(* CODESYS project yaskawafunctions.library
   Company: Evolution
   Title: YaskawaFunctions
   Version: 1.0.0.0

Project tree, tasks and I/O mapping:
  libraries: Tc2_System, * (Beckhoff Automation GmbH); Tc2_Utilities, * (Beckhoff Automation GmbH); Tc2_EtherCAT, * (Beckhoff Automation GmbH); Tc2_Standard, * (Beckhoff Automation GmbH)
  Data types/
    data type E_AccessType
    data type E_AmpType
    data type E_AmpVers
    data type E_EepromType
    data type E_SpecialParameter
    data type E_ValueType
    data type E_WhenEnabled
    data type E_Y_FB_Version
    data type ST_SigmaObject
  Global Variables/
    global variables Constants
  POUs/
    function block Y_AbsoluteEncoderReset [ST]
    function block Y_StoreParameters [ST]
    function block Y_WriteParameters [ST]
  Visualizations/
*)

// Data types/E_AccessType
TYPE E_AccessType : (
	ACCESS_RO		:=0,
	ACCESS_RW	:=1
	);
END_TYPE

// Data types/E_AmpType
TYPE E_AmpType : (
	BOTH_ROT_LIN		:=0,
	ROTARY			:=1,
	LINEAR				:=2
	);
END_TYPE

// Data types/E_AmpVers
TYPE E_AmpVers : (
	VERS_1_0	:=1,
	VERS_2_0	:=2	(*Vers Up*)
	);
END_TYPE

// Data types/E_EepromType
TYPE E_EepromType : (
	EEPROM_NO	:=0,
	EEPROM_YES	:=1
	);
END_TYPE

// Data types/E_SpecialParameter
TYPE E_SpecialParameter : (
	NOTHING_SPECIAL										:=0,	(*	16#0000	*)
	CHANGE_ECAT_PREOP							 		:=1,	(*	16#0001	*)	(*This object can be changed only in the EtherCAT Pre-Operational state*)
	CONDITIONAL_OBJECT									:=2,	(*	16#0002	*)	(*This object has to be set after another object is set. Ex:1C12:01*)
	CHANGE_ECAT_PREOP_AND_IS_DEPENDENT				:=3,
	OBJECT_COMMAND										:=4,	(*	16#0004	*)	(*This object must be executed to enable new settings.  Ex:2700h*)
(*	OBJECT_COMMAND_AND_CHANGE_ECAT_PREOP			:=5,
	OBJECT_COMMAND_AND_IS_DEPENDENT					:=6,
	OBJECT_COMMAND_AND_CHANGE_ECAT_PREOP_AND_IS_DEPENDENT	:=7,
*)	CHANGE_ECAT_DISABLED								:=8,	(*	16#0008	*)	(*This object can be changed only in Switch on Dsiabled state.*)
(*	CHANGE_ECAT_DISABLED_AND_CHANGE_ECAT_PREOP	:=9
	...
*)	CHANGE_ECAT_DISABLED_AND_OBJECT_COMMAND		:=12,	(*	16#0008 OR 16#0004 = 16#000C*)
(*	...
*)	HAS_DEPENDENT										:=16,	(*	16#0010	*)
(*	...
*)	CHANGE_ECAT_PREOP_AND_HAS_DEPENDENT			:=17	(*	16#0010 OR 16#0001 = 16#0011*)	
(*	...
	FUTURE_ADDITION_A									:=32,	(*	16#0020	*)
	...
	FUTURE_ADDITION_B									:=64,	(*	16#0020	*)
	...
*)

	);
END_TYPE

// Data types/E_ValueType
TYPE E_ValueType : (
	TYPE_NOT_SPECIFIED	:=0,
	TYPE_SINT				:=1,
	TYPE_INT				:=2,
	TYPE_DINT				:=3,
	TYPE_USINT			:=4,
	TYPE_UINT				:=5,
	TYPE_UDINT			:=6,
	TYPE_STRING			:=7
	);
END_TYPE

// Data types/E_WhenEnabled
TYPE E_WhenEnabled : (
	ENABLED_IMMEDIATELY		:=0,
	ENABLED_AFTER_RESTART 	:=1,
	ENABLED_SPECIAL			:=2
	);
END_TYPE

// Data types/E_Y_FB_Version
TYPE E_Y_FB_Version : (
	Y_FB_VER_1_0	:=1,
	Y_FB_VER_2_0	:=2	(*Vers Up*)
	);
END_TYPE

// Data types/ST_SigmaObject
TYPE ST_SigmaObject :
STRUCT
	Index			: WORD;		(* Index *)
	SubIndex		: USINT;		(* sub index *)
	(*Data type = UDINT*)
	Access				: USINT;	 	(*ENUM: ACCESS_RW, ACCESS_RO*)
	Eeprom				: USINT;	 	(*ENUM: EEPROM_NO, EEPROM_YES*)
	ValueSint			: SINT;		(* Parameter Data *)
	ValueInt				: INT;		(* Parameter Data *)
	ValueDint			: DINT;		(* Parameter Data *)
	ValueUsint			: USINT;		(* Parameter Data *)
	ValueUint			: UINT;		(* Parameter Data *)
	ValueUdint			: UDINT;		(* Parameter Data *)
	ValueString			: STRING;	(* Parameter Data *)
	ValueType			: USINT;		(*Parameter Data Type*)
	WhenEnabled		: USINT;		(*ENUM: ENABLED_AFTER_RESTART, ENABLED_IMMEDIATELY*)
	AmpType			: USINT; 		(*ENUM: ROTARY, LINEAR, BOTH_ROT_LIN*)
	EnRestartPattern		: WORD;		(* Specifies which bits of the parameter data require restart when changed *)
	AmpVers			: USINT 		:= VERS_1_0;
	SpecialParameter		: DWORD;	(*allows up to 32 switches*)
	DependentValueUsint	: USINT;		(*0 in all cases for version 1, Ex: 1600, 1601...*)

END_STRUCT
END_TYPE

// Global Variables/Constants
{attribute 'Tc2GvlVarNames'}
VAR_GLOBAL CONSTANT
	SAVE				:	UDINT		:=	16#65766173;		(*This is SAVE in ASCII with MSB leftmost, so that's EVAS*)
	USERPRMCFG		:	UDINT		:=	1;
	REVISION_1			:	UDINT		:=	16#00010000;
	REVISION_2			:	UDINT		:=	16#00020000;		(*Vers Up*)
	VENDOR_YASKAWA	:	UDINT		:=	16#00000539;
	PRODUCT_ROTARY	:	UDINT		:=	16#02200001;
	PRODUCT_LINEAR	:	UDINT		:=	16#02200002;
	SEND_REQUEST_1008	:	ARRAY [1..16] OF USINT	:=[	0,0,1,2,00,16#20,0,0,16#08,16#10,0,0,0,0,0,0];
	SEND_REQUEST_100E	:	ARRAY [1..16] OF USINT	:=[	0,0,1,2,00,16#20,0,0,16#0E,16#10,0,0,0,0,0,0];
	SEND_REQUEST_1013	:	ARRAY [1..16] OF USINT	:=[	0,0,1,2,00,16#20,0,0,16#13,16#10,0,0,0,0,0,0];
	SEND_PREPARATION	:	ARRAY [1..16] OF USINT		:=[	0,0,1,2,01,16#20,0,0,16#02,16#00,0,0,0,0,0,0];
	SEND_EXECUTE			:	ARRAY [1..16] OF USINT	:=[	0,0,1,2,01,16#20,0,0,16#01,16#00,0,0,0,0,0,0];
	SEND_ABORT			:	ARRAY [1..16] OF USINT	:=[	0,0,1,2,00,16#20,0,0,16#00,16#00,0,0,0,0,0,0];
END_VAR
VAR_GLOBAL
END_VAR

// POUs/Y_AbsoluteEncoderReset
FUNCTION_BLOCK Y_AbsoluteEncoderReset
VAR_INPUT
	bExecute		:	BOOL		;
	sNetId			:	T_AmsNetId	;
	nSlaveAddr 		:	UINT		;
END_VAR
VAR_OUTPUT
	bDone		:	BOOL			;
	bBusy		:	BOOL			;
	bError		:	BOOL			;
	nErrorID		:	UDINT			;
END_VAR
VAR
(*Extra Features Var Out*)
	sErrorString	:	T_MaxString		;
(*Internal variables*)
	State				:	UINT		:= 	0;
	VendorID			: 	UDINT		;
	ProductCode			: 	UDINT		;
	bNotExecute			:	BOOL		;
	StatusWord			: 	UINT		;
	nErrorIDRead			:	UDINT		;
	sNetIdRead			:	T_AmsNetId	;
	nSlaveAddrRead		:	UINT		;
	StatusAdjusting		:	USINT		;

(*Internal Function Blocks*)
	fbRisingEdge			: 	R_TRIG	;
	fbFallingEdge		: 	F_TRIG	;
	fbSdoReadEx		: 	FB_EcCoESdoReadEx 	:= (bExecute := FALSE, bCompleteAccess := FALSE);
	fbSdoWriteEx			:	FB_EcCoESdoWriteEx 	:= (bExecute := FALSE, bCompleteAccess := FALSE);
END_VAR

fbFallingEdge	(CLK:= bExecute);
IF fbFallingEdge.Q THEN
	bNotExecute	:=	TRUE;
END_IF;

(* Done is TRUE for one cycle when falling edge of Execute has occured *)
IF bDone AND bNotExecute THEN
	bDone		:=	FALSE;
END_IF;

IF bError AND bNotExecute THEN
	bError				:=	FALSE;
	nErrorId				:=	0;
	nErrorIDRead			:=	0;
END_IF;

CASE State OF
0:
fbRisingEdge		(CLK:= bExecute);
IF fbRisingEdge.Q THEN
	bDone				:=	FALSE;
	bBusy				:=	TRUE;
	bError				:=	FALSE;
	nErrorId				:=	0;
	nErrorIDRead			:=	0;
	sErrorString			:=	'';
	bNotExecute			:=	FALSE;
	sNetIdRead			:=	sNetId;
	nSlaveAddrRead		:=	nSlaveAddr;
	State				:=	10;
END_IF

1:
fbSdoReadEx(
	sNetId		:=	sNetIdRead,
	nSlaveAddr	:=	nSlaveAddrRead,
	nIndex		:=	16#1018,
	nSubIndex	:=	1,				(*Vendor ID*)
	pDstBuf		:=	ADR(VendorID),
	cbBufLen	:=	SIZEOF(VendorID),
	bExecute	:=	TRUE	);
State:=2;

2: (*SDO read, Read ID*)
fbSdoReadEx();
IF NOT fbSdoReadEx.bBusy THEN
	IF NOT fbSdoReadEx.bError THEN
		fbSdoReadEx(bExecute:= FALSE);
		State:=3;
		IF NOT (VendorID=VENDOR_YASKAWA) THEN 			(*Vendor ID = Yaskawa*)
			sErrorString:=CONCAT(CONCAT(
				'Product not compatible.  This FB is only for Vendor ID 0x00000539 (Yaskawa).  Vendor ID read as ',
				UDINT_TO_STRING(VendorID)),
				'.  ErrorID from FB, not from ADS.'
			);
			nErrorIDRead:=4100;
			State:=99;
		END_IF
	ELSE
		sErrorString:=CONCAT(CONCAT(
			'Error reading Product Code, Object: ',
			WORD_TO_STRING(fbSdoReadEx.nIndex)),
			'.  Perhaps the Axis Address or NetID is incorrect.  Error occurred using Function Block FB_EcCoESdoReadEx.  ErrorID is from FB_EcCoESdoReadEx.'
		);
		nErrorIDRead:=fbSdoReadEx.nErrId;
		State:=99;
	END_IF
END_IF

3: (*Read the product code*)
fbSdoReadEx(
	nSubIndex	:=	2,				(*Product Code*)
	pDstBuf		:=	ADR(ProductCode),
	cbBufLen	:=	SIZEOF(ProductCode),
	bExecute	:=	TRUE);
State:=4;

4: (*SDO read, Read ID*)
fbSdoReadEx();
IF NOT fbSdoReadEx.bBusy THEN
	IF NOT fbSdoReadEx.bError THEN
		fbSdoReadEx(bExecute:= FALSE);
		IF ProductCode=PRODUCT_ROTARY OR ProductCode=PRODUCT_LINEAR THEN 			(*Rotary Motor Detected*)
			State:=10;
		ELSE 									 (*neither Linear nor Rotary Motor Detected*)
			sErrorString:=CONCAT(CONCAT(
				'Product not compatible.  This FB is only for Product codes 0x02200001 (Sigma-5 Rotary) and 0x02200002 (Sigma-5 Linear).  If using Sigma-5 CoE Drive, get latest FB from Yaskawa.com.  Product code read as ',
				UDINT_TO_STRING(ProductCode)),
				'.  ErrorID from FB, not from ADS.'
			);
			nErrorIDRead:=4101;
			State:=99;
		END_IF
	ELSE
		sErrorString:=CONCAT(CONCAT(
			'Error reading Product Code, Object: ',
			WORD_TO_STRING(fbSdoReadEx.nIndex)),
			'.  Error occurred using Function Block FB_EcCoESdoReadEx.  ErrorID is from FB_EcCoESdoReadEx.'
		);
		nErrorIDRead:=fbSdoReadEx.nErrId;
		State:=99;
	END_IF
END_IF

10: (*check conditions for Absolute Reset - check for servo off - doesn't matter the encoder type, since incremental cannot be checked through ECAT*)
fbSdoReadEx( 			(*Get StatusWord*)
	sNetId		:= sNetIdRead,
	nSlaveAddr	:= nSlaveAddrRead ,
	nSubIndex	:= 0,
	nIndex		:= 16#6041,
	pDstBuf		:= ADR(StatusWord),
	cbBufLen	:= SIZEOF(StatusWord),
	bExecute	:= TRUE 		); (*rising edge required*)
State:=11;

11: (*Read the statusword to verify correct state for sending the adjusting command*)
fbSdoReadEx();
IF NOT fbSdoReadEx.bBusy THEN
	IF NOT fbSdoReadEx.bError THEN
		fbSdoReadEx(bExecute:= FALSE);
		IF
			NOT((UINT_TO_WORD(StatusWord) AND 2#0000_0000_0110_1111)=2#0000_0000_0000_0111) (*NOT Quick stop active*)
			AND
			NOT((UINT_TO_WORD(StatusWord) AND 2#0000_0010_0111_1111)=2#0000_0010_0011_0111) (*NOT Operation enabled*)
			AND
			NOT((UINT_TO_WORD(StatusWord) AND 2#0000_0000_0100_1111)=2#0000_0000_0000_1111) (*NOT Fault reaction active*)
			THEN 	(*servo is off - Required specifically for absolute encoder reset*)
			fbSdoWriteEx( (*Initialize WriteEx*)
				sNetId		:= sNetIdRead,
				nSlaveAddr	:= nSlaveAddrRead,
				bExecute	:= FALSE	); (*Second time initialized - first time was in declarations; maybe this line can be removed*)
			State:=12;
		ELSE
			sErrorString:=CONCAT(CONCAT(
				'Servo is on. StatusWord cannot be x00x_0111(bin), xx1x_x011_0111(bin), or x0xx_1111(bin), but read as ',
				UDINT_TO_STRING(StatusWord)),
				'(dec).  ErrorID from FB, not from ADS.'
			);
			nErrorIDRead:=4110;
			State:=99;
		END_IF
	ELSE
		sErrorString:=CONCAT(CONCAT(
			'Error reading StatusWord, Object: ',
			WORD_TO_STRING(fbSdoReadEx.nIndex)),
			'.  Error occurred using Function Block FB_EcCoESdoReadEx.  ErrorID is from FB_EcCoESdoReadEx.'
		);
		nErrorIDRead:=fbSdoReadEx.nErrId;
		State:=99;
	END_IF
END_IF

12: (*Send the data for the Request*)
fbSdoWriteEx(
	nIndex		:= 16#2710,
	nSubIndex	:= 1,
	pSrcBuf		:= ADR(SEND_REQUEST_1008), (*Absolute encoder reset*)
	cbBufLen	:= SIZEOF(SEND_REQUEST_1008),
	bExecute	:= TRUE);
State:=13;

13: (*Complete sending the request*)
fbSdoWriteEx();
IF NOT fbSdoWriteEx.bBusy THEN
	IF NOT fbSdoWriteEx.bError THEN
		fbSdoWriteEx(bExecute:= FALSE);
		State:=14;
	ELSE
		sErrorString:='Error sending Absolute Encoder Reset request to object 2710.  Error occurred using Function Block FB_EcCoESdoWriteEx.  ErrorID is from FB_EcCoESdoWriteEx.';
		nErrorIDRead:=fbSdoWriteEx.nErrId;
		State:=99;
	END_IF
END_IF

14:
fbSdoReadEx( 			(*Get Status (from 2710:02 USINT)*)
	nSubIndex	:= 2,
	nIndex		:= 16#2710,
	pDstBuf		:= ADR(StatusAdjusting),
	cbBufLen	:= SIZEOF(StatusAdjusting),
	bExecute	:= TRUE);
State:=15;

15: (*Read the Status to determine which state to perform next*)
fbSdoReadEx();
IF NOT fbSdoReadEx.bBusy THEN
	IF NOT fbSdoReadEx.bError THEN
		fbSdoReadEx(bExecute:= FALSE);
		CASE StatusAdjusting OF
			1:
				State:=20;
			2:	(*Error. Issue error, then issue Send Abort*)
				sErrorString:='Adjusting command: Send Request 1008 - failed.';
				nErrorIDRead:=4115;
				State:=50;
			3: 	(*Error. Read reply, Issue error, then issue Send Abort*)
				sErrorString:='Adjusting command: Send Request 1008 - failed.  Reply data exists in 0x2710:03.';
				nErrorIDRead:=4116;
				State:=50;
			255:
				State:=14;
			ELSE
				sErrorString:=CONCAT(CONCAT(
					'Status state is not valid (must be 1,2,3,255).  Read as ',
					UDINT_TO_STRING(StatusAdjusting)),
					'(dec).  ErrorID from FB, not from ADS.'
				);
				nErrorIDRead:=4111;
				State:=99;
			END_CASE
	ELSE
		sErrorString:='Error reading Adjusting Status, Object 2710:02.  Error occurred using Function Block FB_EcCoESdoReadEx.  ErrorID is from FB_EcCoESdoReadEx.';
		nErrorIDRead:=fbSdoReadEx.nErrId;
		State:=99;
	END_IF
END_IF

20: (*Continue with Step 2: Send the Preparation*)
(*Preparation is required for Absolute Encoder Reset*)
(*Send the data for the Preparation*)
fbSdoWriteEx(
	nIndex		:= 16#2710,
	nSubIndex	:= 1,
	pSrcBuf		:= ADR(SEND_PREPARATION),
	cbBufLen	:= SIZEOF(SEND_PREPARATION),
	bExecute	:= TRUE);
State:=21;

21: (*Complete sending the request*)
fbSdoWriteEx();
IF NOT fbSdoWriteEx.bBusy THEN
	IF NOT fbSdoWriteEx.bError THEN
		fbSdoWriteEx(bExecute:= FALSE);
		State:=22;
	ELSE
		sErrorString:='Error sending Preparation request to object 2710.  Error occurred using Function Block FB_EcCoESdoWriteEx.  ErrorID is from FB_EcCoESdoWriteEx.';
		nErrorIDRead:=fbSdoWriteEx.nErrId;
		State:=99;
	END_IF
END_IF

22:
fbSdoReadEx( 			(*Get Status (from 2710:02 USINT)*)
	nSubIndex	:= 2,
	nIndex		:= 16#2710,
	pDstBuf		:= ADR(StatusAdjusting),
	cbBufLen	:= SIZEOF(StatusAdjusting),
	bExecute	:= TRUE);
State:=23;

23: (*Read the Status to determine which state to perform next*)
fbSdoReadEx();
IF NOT fbSdoReadEx.bBusy THEN
	IF NOT fbSdoReadEx.bError THEN
		fbSdoReadEx(bExecute:= FALSE);
		CASE StatusAdjusting OF
			1:
				State:=30;
			2:	(*Error. Issue error, then issue Send Abort*)
				sErrorString:='Adjusting command: Send Preparation - failed.';
				nErrorIDRead:=4117;
				State:=50;
			3: 	(*Error. Read reply, Issue error, then issue Send Abort*)
				sErrorString:='Adjusting command: Send Preparation - failed.  Reply data exists in 0x2710:03.';
				nErrorIDRead:=4118;
				State:=50;
			255:
				State:=22;
			ELSE
				sErrorString:=CONCAT(CONCAT(
					'Status state is not valid (must be 1,2,3,255).  Read as ',
					UDINT_TO_STRING(StatusAdjusting)),
					'(dec).  ErrorID from FB, not from ADS.'
				);
				nErrorIDRead:=4111;
				State:=99;
			END_CASE
	ELSE
		sErrorString:='Error reading Adjusting Status, Object 2710:02.  Error occurred using Function Block FB_EcCoESdoReadEx.  ErrorID is from FB_EcCoESdoReadEx.';
		nErrorIDRead:=fbSdoReadEx.nErrId;
		State:=99;
	END_IF
END_IF

30: (*Continue with Step 2: Send the Execute*)
(*Send the data for the Execute*)
fbSdoWriteEx(
	nIndex		:= 16#2710,
	nSubIndex	:= 1,
	pSrcBuf		:= ADR(SEND_EXECUTE),
	cbBufLen	:= SIZEOF(SEND_EXECUTE),
	bExecute	:= TRUE);
State:=31;

31: (*Complete sending the request*)
fbSdoWriteEx();
IF NOT fbSdoWriteEx.bBusy THEN
	IF NOT fbSdoWriteEx.bError THEN
		fbSdoWriteEx(bExecute:= FALSE);
		State:=32;
	ELSE
		sErrorString:='Error sending Execute request to object 2710.  Error occurred using Function Block FB_EcCoESdoWriteEx.  ErrorID is from FB_EcCoESdoWriteEx.';
		nErrorIDRead:=fbSdoWriteEx.nErrId;
		State:=99;
	END_IF
END_IF

32:
fbSdoReadEx( 			(*Get Status (from 2710:02 USINT)*)
	nSubIndex	:= 2,
	nIndex		:= 16#2710,
	pDstBuf		:= ADR(StatusAdjusting),
	cbBufLen	:= SIZEOF(StatusAdjusting),
	bExecute	:= TRUE);
State:=33;

33: (*Read the Status to determine which state to perform next*)
fbSdoReadEx();
IF NOT fbSdoReadEx.bBusy THEN
	IF NOT fbSdoReadEx.bError THEN
		fbSdoReadEx(bExecute:= FALSE);
		CASE StatusAdjusting OF
			1:
				State:=40;
			2:	(*Error. Issue error, then issue Send Abort*)
				sErrorString:='Adjusting command: Send Execute - failed.';
				nErrorIDRead:=4119;
				State:=50;
			3: 	(*Error. Read reply, Issue error, then issue Send Abort*)
				sErrorString:='Adjusting command: Send Execute - failed.  Reply data exists in 0x2710:03.';
				nErrorIDRead:=4120;
				State:=50;
			255:
				State:=32;
			ELSE
				sErrorString:=CONCAT(CONCAT(
					'Status state is not valid (must be 1,2,3,255).  Read as ',
					UDINT_TO_STRING(StatusAdjusting)),
					'(dec).  ErrorID from FB, not from ADS.'
				);
				nErrorIDRead:=4111;
				State:=99;
			END_CASE
	ELSE
		sErrorString:='Error reading Adjusting Status, Object 2710:02.  Error occurred using Function Block FB_EcCoESdoReadEx.  ErrorID is from FB_EcCoESdoReadEx.';
		nErrorIDRead:=fbSdoReadEx.nErrId;
		State:=99;
	END_IF
END_IF

40: (*Finished Execution*)
	bDone	:=	TRUE;
	bBusy	:=	FALSE;
	State:=0;

50: (*Step 4: Send Abort (only applies if an error occurs)*)
fbSdoWriteEx(
	nIndex		:= 16#2710,
	nSubIndex	:= 1,
	pSrcBuf		:= ADR(SEND_ABORT),
	cbBufLen	:= SIZEOF(SEND_ABORT),
	bExecute	:= TRUE);
State:=51;

51: (*Complete sending the request*)
fbSdoWriteEx();
IF NOT fbSdoWriteEx.bBusy THEN
	IF NOT fbSdoWriteEx.bError THEN
		fbSdoWriteEx(bExecute:= FALSE);
		State:=52;
	ELSE
		sErrorString:='Error sending Abort request to object 2710.  Error occurred using Function Block FB_EcCoESdoWriteEx.  ErrorID is from FB_EcCoESdoWriteEx.  Also, error occurred performing Adjusting command, but ErrorID of this second error cannot be provided.';
		nErrorIDRead:=fbSdoWriteEx.nErrId;
		State:=99;
	END_IF
END_IF

52:
fbSdoReadEx( 			(*Get Status (from 2710:02 USINT)*)
	nSubIndex	:= 2,
	nIndex		:= 16#2710,
	pDstBuf		:= ADR(StatusAdjusting),
	cbBufLen	:= SIZEOF(StatusAdjusting),
	bExecute	:= TRUE);
State:=53;

53: (*Read the Status to determine which state to perform next*)
fbSdoReadEx();
IF NOT fbSdoReadEx.bBusy THEN
	IF NOT fbSdoReadEx.bError THEN
		fbSdoReadEx(bExecute:= FALSE);
		CASE StatusAdjusting OF
			1:
				sErrorString:=CONCAT(
				sErrorString,  (*Concatenate with error string from previous error state.*)
				'  Abort succeeded, but requested adjusting command failed.  ErrorID is from FB, not from ADS.'
				);
				State:=99;
			2:
				sErrorString:='Abort failed, and requested adjusting command failed.  ErrorID is from FB, not from ADS.';
				nErrorIDRead:=4113;
				State:=99;
			3:
				sErrorString:='Abort failed, and requested adjusting command failed.  Reply data exists in 0x2710:03.  ErrorID is from FB, not from ADS.';
				nErrorIDRead:=4114;
				State:=99;
			255:
				State:=52;
			ELSE
				sErrorString:=CONCAT(CONCAT(
					'Status state is not valid (must be 1,2,3,255).  Read as ',
					UDINT_TO_STRING(StatusAdjusting)),
					'(dec).  ErrorID from FB, not from ADS.  Also, error occurred performing Adjusting command, but ErrorID of this second error cannot be provided.'
				);
				nErrorIDRead:=4111;
				State:=99;
			END_CASE
	ELSE
		sErrorString:='Error reading Adjusting Status, Object 2710:02.  Error occurred using Function Block FB_EcCoESdoReadEx.  ErrorID is from FB_EcCoESdoReadEx.  Also, error occurred performing Adjusting command, but ErrorID of this second error cannot be provided.';
		nErrorIDRead:=fbSdoReadEx.nErrId;
		State:=99;
	END_IF
END_IF

99: (*Error State*)
	bBusy	:=	FALSE;
	bError	:=	TRUE;
	nErrorID	:=	nErrorIDRead;
	State	:=	0;

ELSE
	sErrorString:=CONCAT(CONCAT(
		'Internal function block error.  Function block state not found.  State read as: ',
		UINT_TO_STRING(State)),
		'.  ErrorID from FB, not from ADS.'
	);
	nErrorIDRead:=4112;
	State:=99;
END_CASE

END_FUNCTION_BLOCK

// POUs/Y_StoreParameters
FUNCTION_BLOCK Y_StoreParameters
VAR_INPUT
	bExecute		:	BOOL		;
	sNetId			:	T_AmsNetId	;
	nSlaveAddr 		:	UINT		;
	sFile			:	T_MaxString	:=	'C:\YaskawaPrm.dat' ;
END_VAR
VAR_OUTPUT
	bDone		:	BOOL			;
	bBusy		:	BOOL			;
	bError		:	BOOL			;
	nErrorID		:	UDINT			;
END_VAR
VAR
	(*Extra Features Var In*)
	bBypassCheck	:	BOOL		:=	FALSE;					(*Used to skip Version check, but not Vendor ID nor Product Code*)
	bBypassAutoFile	:	BOOL		:=	TRUE;
	sFileAuto		:	T_MaxString	:=	'C:\YaskawaPrm_'	; (*Time stamp and .dat is appended to this file name*)
	(*Extra Features Var Out*)
	sErrorString	:	T_MaxString		;

	AllSigmaObjects : ARRAY [1..364] OF ST_SigmaObject:=[
(*1*)		(Index:=16#1000,	SubIndex:=0,		ValueType:=TYPE_UDINT,		Access:=ACCESS_RO,		Eeprom:=EEPROM_NO,	AmpType:=BOTH_ROT_LIN,	WhenEnabled:=ENABLED_IMMEDIATELY),
		(Index:=16#1001,	SubIndex:=0,		ValueType:=TYPE_USINT,		Access:=ACCESS_RO,		Eeprom:=EEPROM_NO,	AmpType:=BOTH_ROT_LIN,	WhenEnabled:=ENABLED_IMMEDIATELY),
		(Index:=16#1008,	SubIndex:=0,		ValueType:=TYPE_STRING,	Access:=ACCESS_RO,		Eeprom:=EEPROM_NO,	AmpType:=BOTH_ROT_LIN,	WhenEnabled:=ENABLED_IMMEDIATELY),
		(Index:=16#100A,	SubIndex:=0,		ValueType:=TYPE_STRING,	Access:=ACCESS_RO,		Eeprom:=EEPROM_NO,	AmpType:=BOTH_ROT_LIN,	WhenEnabled:=ENABLED_IMMEDIATELY),
		(Index:=16#1010,	SubIndex:=0,		ValueType:=TYPE_USINT,		Access:=ACCESS_RO,		Eeprom:=EEPROM_NO,	AmpType:=BOTH_ROT_LIN,	WhenEnabled:=ENABLED_IMMEDIATELY),
		(Index:=16#1010,	SubIndex:=1,		ValueType:=TYPE_UDINT,		Access:=ACCESS_RW,	Eeprom:=EEPROM_NO,	AmpType:=BOTH_ROT_LIN,	WhenEnabled:=ENABLED_IMMEDIATELY,		SpecialParameter:=CHANGE_ECAT_DISABLED_AND_OBJECT_COMMAND),
		(Index:=16#1010,	SubIndex:=2,		ValueType:=TYPE_UDINT,		Access:=ACCESS_RW,	Eeprom:=EEPROM_NO,	AmpType:=BOTH_ROT_LIN,	WhenEnabled:=ENABLED_IMMEDIATELY,		SpecialParameter:=OBJECT_COMMAND),
		(Index:=16#1010,	SubIndex:=3,		ValueType:=TYPE_UDINT,		Access:=ACCESS_RW,	Eeprom:=EEPROM_NO,	AmpType:=BOTH_ROT_LIN,	WhenEnabled:=ENABLED_IMMEDIATELY,		SpecialParameter:=OBJECT_COMMAND),
		(Index:=16#1010,	SubIndex:=4,		ValueType:=TYPE_UDINT,		Access:=ACCESS_RW,	Eeprom:=EEPROM_NO,	AmpType:=BOTH_ROT_LIN,	WhenEnabled:=ENABLED_IMMEDIATELY,		SpecialParameter:=CHANGE_ECAT_DISABLED_AND_OBJECT_COMMAND),
(*10*)	(Index:=16#1011,	SubIndex:=0,		ValueType:=TYPE_USINT,		Access:=ACCESS_RO,		Eeprom:=EEPROM_NO,	AmpType:=BOTH_ROT_LIN,	WhenEnabled:=ENABLED_IMMEDIATELY),
		(Index:=16#1011,	SubIndex:=1,		ValueType:=TYPE_UDINT,		Access:=ACCESS_RW,	Eeprom:=EEPROM_NO,	AmpType:=BOTH_ROT_LIN,	WhenEnabled:=ENABLED_IMMEDIATELY,		SpecialParameter:=CHANGE_ECAT_DISABLED_AND_OBJECT_COMMAND),
		(Index:=16#1011,	SubIndex:=2,		ValueType:=TYPE_UDINT,		Access:=ACCESS_RW,	Eeprom:=EEPROM_NO,	AmpType:=BOTH_ROT_LIN,	WhenEnabled:=ENABLED_IMMEDIATELY,		SpecialParameter:=OBJECT_COMMAND),
		(Index:=16#1011,	SubIndex:=3,		ValueType:=TYPE_UDINT,		Access:=ACCESS_RW,	Eeprom:=EEPROM_NO,	AmpType:=BOTH_ROT_LIN,	WhenEnabled:=ENABLED_IMMEDIATELY,		SpecialParameter:=OBJECT_COMMAND),
		(Index:=16#1011,	SubIndex:=4,		ValueType:=TYPE_UDINT,		Access:=ACCESS_RW,	Eeprom:=EEPROM_NO,	AmpType:=BOTH_ROT_LIN,	WhenEnabled:=ENABLED_IMMEDIATELY,		SpecialParameter:=CHANGE_ECAT_DISABLED_AND_OBJECT_COMMAND),
		(Index:=16#1018,	SubIndex:=0,		ValueType:=TYPE_USINT,		Access:=ACCESS_RO,		Eeprom:=EEPROM_NO,	AmpType:=BOTH_ROT_LIN,	WhenEnabled:=ENABLED_IMMEDIATELY),
		(Index:=16#1018,	SubIndex:=1,		ValueType:=TYPE_UDINT,		Access:=ACCESS_RO,		Eeprom:=EEPROM_NO,	AmpType:=BOTH_ROT_LIN,	WhenEnabled:=ENABLED_IMMEDIATELY),
		(Index:=16#1018,	SubIndex:=2,		ValueType:=TYPE_UDINT,		Access:=ACCESS_RO,		Eeprom:=EEPROM_NO,	AmpType:=BOTH_ROT_LIN,	WhenEnabled:=ENABLED_IMMEDIATELY),
		(Index:=16#1018,	SubIndex:=3,		ValueType:=TYPE_UDINT,		Access:=ACCESS_RO,		Eeprom:=EEPROM_NO,	AmpType:=BOTH_ROT_LIN,	WhenEnabled:=ENABLED_IMMEDIATELY),
		(Index:=16#1018,	SubIndex:=4,		ValueType:=TYPE_UDINT,		Access:=ACCESS_RO,		Eeprom:=EEPROM_NO,	AmpType:=BOTH_ROT_LIN,	WhenEnabled:=ENABLED_IMMEDIATELY),
(*20*)	(Index:=16#1600,	SubIndex:=0,		ValueType:=TYPE_USINT,		Access:=ACCESS_RW,	Eeprom:=EEPROM_YES,	AmpType:=BOTH_ROT_LIN,	WhenEnabled:=ENABLED_IMMEDIATELY,		SpecialParameter:=CHANGE_ECAT_PREOP_AND_HAS_DEPENDENT,		DependentValueUsint:=0),
		(Index:=16#1600,	SubIndex:=1,		ValueType:=TYPE_UDINT,		Access:=ACCESS_RW,	Eeprom:=EEPROM_YES,	AmpType:=BOTH_ROT_LIN,	WhenEnabled:=ENABLED_IMMEDIATELY,		SpecialParameter:=CHANGE_ECAT_PREOP_AND_IS_DEPENDENT),
		(Index:=16#1600,	SubIndex:=2,		ValueType:=TYPE_UDINT,		Access:=ACCESS_RW,	Eeprom:=EEPROM_YES,	AmpType:=BOTH_ROT_LIN,	WhenEnabled:=ENABLED_IMMEDIATELY,		SpecialParameter:=CHANGE_ECAT_PREOP_AND_IS_DEPENDENT),
		(Index:=16#1600,	SubIndex:=3,		ValueType:=TYPE_UDINT,		Access:=ACCESS_RW,	Eeprom:=EEPROM_YES,	AmpType:=BOTH_ROT_LIN,	WhenEnabled:=ENABLED_IMMEDIATELY,		SpecialParameter:=CHANGE_ECAT_PREOP_AND_IS_DEPENDENT),
		(Index:=16#1600,	SubIndex:=4,		ValueType:=TYPE_UDINT,		Access:=ACCESS_RW,	Eeprom:=EEPROM_YES,	AmpType:=BOTH_ROT_LIN,	WhenEnabled:=ENABLED_IMMEDIATELY,		SpecialParameter:=CHANGE_ECAT_PREOP_AND_IS_DEPENDENT),
		(Index:=16#1600,	SubIndex:=5,		ValueType:=TYPE_UDINT,		Access:=ACCESS_RW,	Eeprom:=EEPROM_YES,	AmpType:=BOTH_ROT_LIN,	WhenEnabled:=ENABLED_IMMEDIATELY,		SpecialParameter:=CHANGE_ECAT_PREOP_AND_IS_DEPENDENT),
		(Index:=16#1600,	SubIndex:=6,		ValueType:=TYPE_UDINT,		Access:=ACCESS_RW,	Eeprom:=EEPROM_YES,	AmpType:=BOTH_ROT_LIN,	WhenEnabled:=ENABLED_IMMEDIATELY,		SpecialParameter:=CHANGE_ECAT_PREOP_AND_IS_DEPENDENT),
		(Index:=16#1600,	SubIndex:=7,		ValueType:=TYPE_UDINT,		Access:=ACCESS_RW,	Eeprom:=EEPROM_YES,	AmpType:=BOTH_ROT_LIN,	WhenEnabled:=ENABLED_IMMEDIATELY,		SpecialParameter:=CHANGE_ECAT_PREOP_AND_IS_DEPENDENT),
		(Index:=16#1600,	SubIndex:=8,		ValueType:=TYPE_UDINT,		Access:=ACCESS_RW,	Eeprom:=EEPROM_YES,	AmpType:=BOTH_ROT_LIN,	WhenEnabled:=ENABLED_IMMEDIATELY,		SpecialParameter:=CHANGE_ECAT_PREOP_AND_IS_DEPENDENT),
		(Index:=16#1601,	SubIndex:=0,		ValueType:=TYPE_USINT,		Access:=ACCESS_RW,	Eeprom:=EEPROM_YES,	AmpType:=BOTH_ROT_LIN,	WhenEnabled:=ENABLED_IMMEDIATELY,		SpecialParameter:=CHANGE_ECAT_PREOP_AND_HAS_DEPENDENT,		DependentValueUsint:=0),
(*30*)	(Index:=16#1601,	SubIndex:=1,		ValueType:=TYPE_UDINT,		Access:=ACCESS_RW,	Eeprom:=EEPROM_YES,	AmpType:=BOTH_ROT_LIN,	WhenEnabled:=ENABLED_IMMEDIATELY,		SpecialParameter:=CHANGE_ECAT_PREOP_AND_IS_DEPENDENT),
		(Index:=16#1601,	SubIndex:=2,		ValueType:=TYPE_UDINT,		Access:=ACCESS_RW,	Eeprom:=EEPROM_YES,	AmpType:=BOTH_ROT_LIN,	WhenEnabled:=ENABLED_IMMEDIATELY,		SpecialParameter:=CHANGE_ECAT_PREOP_AND_IS_DEPENDENT),
		(Index:=16#1601,	SubIndex:=3,		ValueType:=TYPE_UDINT,		Access:=ACCESS_RW,	Eeprom:=EEPROM_YES,	AmpType:=BOTH_ROT_LIN,	WhenEnabled:=ENABLED_IMMEDIATELY,		SpecialParameter:=CHANGE_ECAT_PREOP_AND_IS_DEPENDENT),
		(Index:=16#1601,	SubIndex:=4,		ValueType:=TYPE_UDINT,		Access:=ACCESS_RW,	Eeprom:=EEPROM_YES,	AmpType:=BOTH_ROT_LIN,	WhenEnabled:=ENABLED_IMMEDIATELY,		SpecialParameter:=CHANGE_ECAT_PREOP_AND_IS_DEPENDENT),
		(Index:=16#1601,	SubIndex:=5,		ValueType:=TYPE_UDINT,		Access:=ACCESS_RW,	Eeprom:=EEPROM_YES,	AmpType:=BOTH_ROT_LIN,	WhenEnabled:=ENABLED_IMMEDIATELY,		SpecialParameter:=CHANGE_ECAT_PREOP_AND_IS_DEPENDENT),
		(Index:=16#1601,	SubIndex:=6,		ValueType:=TYPE_UDINT,		Access:=ACCESS_RW,	Eeprom:=EEPROM_YES,	AmpType:=BOTH_ROT_LIN,	WhenEnabled:=ENABLED_IMMEDIATELY,		SpecialParameter:=CHANGE_ECAT_PREOP_AND_IS_DEPENDENT),
		(Index:=16#1601,	SubIndex:=7,		ValueType:=TYPE_UDINT,		Access:=ACCESS_RW,	Eeprom:=EEPROM_YES,	AmpType:=BOTH_ROT_LIN,	WhenEnabled:=ENABLED_IMMEDIATELY,		SpecialParameter:=CHANGE_ECAT_PREOP_AND_IS_DEPENDENT),
		(Index:=16#1601,	SubIndex:=8,		ValueType:=TYPE_UDINT,		Access:=ACCESS_RW,	Eeprom:=EEPROM_YES,	AmpType:=BOTH_ROT_LIN,	WhenEnabled:=ENABLED_IMMEDIATELY,		SpecialParameter:=CHANGE_ECAT_PREOP_AND_IS_DEPENDENT),
		(Index:=16#1602,	SubIndex:=0,		ValueType:=TYPE_USINT,		Access:=ACCESS_RW,	Eeprom:=EEPROM_YES,	AmpType:=BOTH_ROT_LIN,	WhenEnabled:=ENABLED_IMMEDIATELY,		SpecialParameter:=CHANGE_ECAT_PREOP_AND_HAS_DEPENDENT,		DependentValueUsint:=0),
		(Index:=16#1602,	SubIndex:=1,		ValueType:=TYPE_UDINT,		Access:=ACCESS_RW,	Eeprom:=EEPROM_YES,	AmpType:=BOTH_ROT_LIN,	WhenEnabled:=ENABLED_IMMEDIATELY,		SpecialParameter:=CHANGE_ECAT_PREOP_AND_IS_DEPENDENT),
(*40*)	(Index:=16#1602,	SubIndex:=2,		ValueType:=TYPE_UDINT,		Access:=ACCESS_RW,	Eeprom:=EEPROM_YES,	AmpType:=BOTH_ROT_LIN,	WhenEnabled:=ENABLED_IMMEDIATELY,		SpecialParameter:=CHANGE_ECAT_PREOP_AND_IS_DEPENDENT),
		(Index:=16#1602,	SubIndex:=3,		ValueType:=TYPE_UDINT,		Access:=ACCESS_RW,	Eeprom:=EEPROM_YES,	AmpType:=BOTH_ROT_LIN,	WhenEnabled:=ENABLED_IMMEDIATELY,		SpecialParameter:=CHANGE_ECAT_PREOP_AND_IS_DEPENDENT),
		(Index:=16#1602,	SubIndex:=4,		ValueType:=TYPE_UDINT,		Access:=ACCESS_RW,	Eeprom:=EEPROM_YES,	AmpType:=BOTH_ROT_LIN,	WhenEnabled:=ENABLED_IMMEDIATELY,		SpecialParameter:=CHANGE_ECAT_PREOP_AND_IS_DEPENDENT),
		(Index:=16#1602,	SubIndex:=5,		ValueType:=TYPE_UDINT,		Access:=ACCESS_RW,	Eeprom:=EEPROM_YES,	AmpType:=BOTH_ROT_LIN,	WhenEnabled:=ENABLED_IMMEDIATELY,		SpecialParameter:=CHANGE_ECAT_PREOP_AND_IS_DEPENDENT),
		(Index:=16#1602,	SubIndex:=6,		ValueType:=TYPE_UDINT,		Access:=ACCESS_RW,	Eeprom:=EEPROM_YES,	AmpType:=BOTH_ROT_LIN,	WhenEnabled:=ENABLED_IMMEDIATELY,		SpecialParameter:=CHANGE_ECAT_PREOP_AND_IS_DEPENDENT),
		(Index:=16#1602,	SubIndex:=7,		ValueType:=TYPE_UDINT,		Access:=ACCESS_RW,	Eeprom:=EEPROM_YES,	AmpType:=BOTH_ROT_LIN,	WhenEnabled:=ENABLED_IMMEDIATELY,		SpecialParameter:=CHANGE_ECAT_PREOP_AND_IS_DEPENDENT),
		(Index:=16#1602,	SubIndex:=8,		ValueType:=TYPE_UDINT,		Access:=ACCESS_RW,	Eeprom:=EEPROM_YES,	AmpType:=BOTH_ROT_LIN,	WhenEnabled:=ENABLED_IMMEDIATELY,		SpecialParameter:=CHANGE_ECAT_PREOP_AND_IS_DEPENDENT),
		(Index:=16#1603,	SubIndex:=0,		ValueType:=TYPE_USINT,		Access:=ACCESS_RW,	Eeprom:=EEPROM_YES,	AmpType:=BOTH_ROT_LIN,	WhenEnabled:=ENABLED_IMMEDIATELY,		SpecialParameter:=CHANGE_ECAT_PREOP_AND_HAS_DEPENDENT,		DependentValueUsint:=0),
		(Index:=16#1603,	SubIndex:=1,		ValueType:=TYPE_UDINT,		Access:=ACCESS_RW,	Eeprom:=EEPROM_YES,	AmpType:=BOTH_ROT_LIN,	WhenEnabled:=ENABLED_IMMEDIATELY,		SpecialParameter:=CHANGE_ECAT_PREOP_AND_IS_DEPENDENT),
		(Index:=16#1603,	SubIndex:=2,		ValueType:=TYPE_UDINT,		Access:=ACCESS_RW,	Eeprom:=EEPROM_YES,	AmpType:=BOTH_ROT_LIN,	WhenEnabled:=ENABLED_IMMEDIATELY,		SpecialParameter:=CHANGE_ECAT_PREOP_AND_IS_DEPENDENT),
(*50*)	(Index:=16#1603,	SubIndex:=3,		ValueType:=TYPE_UDINT,		Access:=ACCESS_RW,	Eeprom:=EEPROM_YES,	AmpType:=BOTH_ROT_LIN,	WhenEnabled:=ENABLED_IMMEDIATELY,		SpecialParameter:=CHANGE_ECAT_PREOP_AND_IS_DEPENDENT),
		(Index:=16#1603,	SubIndex:=4,		ValueType:=TYPE_UDINT,		Access:=ACCESS_RW,	Eeprom:=EEPROM_YES,	AmpType:=BOTH_ROT_LIN,	WhenEnabled:=ENABLED_IMMEDIATELY,		SpecialParameter:=CHANGE_ECAT_PREOP_AND_IS_DEPENDENT),
		(Index:=16#1603,	SubIndex:=5,		ValueType:=TYPE_UDINT,		Access:=ACCESS_RW,	Eeprom:=EEPROM_YES,	AmpType:=BOTH_ROT_LIN,	WhenEnabled:=ENABLED_IMMEDIATELY,		SpecialParameter:=CHANGE_ECAT_PREOP_AND_IS_DEPENDENT),
		(Index:=16#1603,	SubIndex:=6,		ValueType:=TYPE_UDINT,		Access:=ACCESS_RW,	Eeprom:=EEPROM_YES,	AmpType:=BOTH_ROT_LIN,	WhenEnabled:=ENABLED_IMMEDIATELY,		SpecialParameter:=CHANGE_ECAT_PREOP_AND_IS_DEPENDENT),
		(Index:=16#1603,	SubIndex:=7,		ValueType:=TYPE_UDINT,		Access:=ACCESS_RW,	Eeprom:=EEPROM_YES,	AmpType:=BOTH_ROT_LIN,	WhenEnabled:=ENABLED_IMMEDIATELY,		SpecialParameter:=CHANGE_ECAT_PREOP_AND_IS_DEPENDENT),
		(Index:=16#1603,	SubIndex:=8,		ValueType:=TYPE_UDINT,		Access:=ACCESS_RW,	Eeprom:=EEPROM_YES,	AmpType:=BOTH_ROT_LIN,	WhenEnabled:=ENABLED_IMMEDIATELY,		SpecialParameter:=CHANGE_ECAT_PREOP_AND_IS_DEPENDENT),
		(Index:=16#1A00,	SubIndex:=0,		ValueType:=TYPE_USINT,		Access:=ACCESS_RW,	Eeprom:=EEPROM_YES,	AmpType:=BOTH_ROT_LIN,	WhenEnabled:=ENABLED_IMMEDIATELY,		SpecialParameter:=CHANGE_ECAT_PREOP_AND_HAS_DEPENDENT,		DependentValueUsint:=0),
		(Index:=16#1A00,	SubIndex:=1,		ValueType:=TYPE_UDINT,		Access:=ACCESS_RW,	Eeprom:=EEPROM_YES,	AmpType:=BOTH_ROT_LIN,	WhenEnabled:=ENABLED_IMMEDIATELY,		SpecialParameter:=CHANGE_ECAT_PREOP_AND_IS_DEPENDENT),
		(Index:=16#1A00,	SubIndex:=2,		ValueType:=TYPE_UDINT,		Access:=ACCESS_RW,	Eeprom:=EEPROM_YES,	AmpType:=BOTH_ROT_LIN,	WhenEnabled:=ENABLED_IMMEDIATELY,		SpecialParameter:=CHANGE_ECAT_PREOP_AND_IS_DEPENDENT),
		(Index:=16#1A00,	SubIndex:=3,		ValueType:=TYPE_UDINT,		Access:=ACCESS_RW,	Eeprom:=EEPROM_YES,	AmpType:=BOTH_ROT_LIN,	WhenEnabled:=ENABLED_IMMEDIATELY,		SpecialParameter:=CHANGE_ECAT_PREOP_AND_IS_DEPENDENT),
(*60*)	(Index:=16#1A00,	SubIndex:=4,		ValueType:=TYPE_UDINT,		Access:=ACCESS_RW,	Eeprom:=EEPROM_YES,	AmpType:=BOTH_ROT_LIN,	WhenEnabled:=ENABLED_IMMEDIATELY,		SpecialParameter:=CHANGE_ECAT_PREOP_AND_IS_DEPENDENT),
		(Index:=16#1A00,	SubIndex:=5,		ValueType:=TYPE_UDINT,		Access:=ACCESS_RW,	Eeprom:=EEPROM_YES,	AmpType:=BOTH_ROT_LIN,	WhenEnabled:=ENABLED_IMMEDIATELY,		SpecialParameter:=CHANGE_ECAT_PREOP_AND_IS_DEPENDENT),
		(Index:=16#1A00,	SubIndex:=6,		ValueType:=TYPE_UDINT,		Access:=ACCESS_RW,	Eeprom:=EEPROM_YES,	AmpType:=BOTH_ROT_LIN,	WhenEnabled:=ENABLED_IMMEDIATELY,		SpecialParameter:=CHANGE_ECAT_PREOP_AND_IS_DEPENDENT),
		(Index:=16#1A00,	SubIndex:=7,		ValueType:=TYPE_UDINT,		Access:=ACCESS_RW,	Eeprom:=EEPROM_YES,	AmpType:=BOTH_ROT_LIN,	WhenEnabled:=ENABLED_IMMEDIATELY,		SpecialParameter:=CHANGE_ECAT_PREOP_AND_IS_DEPENDENT),
		(Index:=16#1A00,	SubIndex:=8,		ValueType:=TYPE_UDINT,		Access:=ACCESS_RW,	Eeprom:=EEPROM_YES,	AmpType:=BOTH_ROT_LIN,	WhenEnabled:=ENABLED_IMMEDIATELY,		SpecialParameter:=CHANGE_ECAT_PREOP_AND_IS_DEPENDENT),
		(Index:=16#1A01,	SubIndex:=0,		ValueType:=TYPE_USINT,		Access:=ACCESS_RW,	Eeprom:=EEPROM_YES,	AmpType:=BOTH_ROT_LIN,	WhenEnabled:=ENABLED_IMMEDIATELY,		SpecialParameter:=CHANGE_ECAT_PREOP_AND_HAS_DEPENDENT,		DependentValueUsint:=0),
		(Index:=16#1A01,	SubIndex:=1,		ValueType:=TYPE_UDINT,		Access:=ACCESS_RW,	Eeprom:=EEPROM_YES,	AmpType:=BOTH_ROT_LIN,	WhenEnabled:=ENABLED_IMMEDIATELY,		SpecialParameter:=CHANGE_ECAT_PREOP_AND_IS_DEPENDENT),
		(Index:=16#1A01,	SubIndex:=2,		ValueType:=TYPE_UDINT,		Access:=ACCESS_RW,	Eeprom:=EEPROM_YES,	AmpType:=BOTH_ROT_LIN,	WhenEnabled:=ENABLED_IMMEDIATELY,		SpecialParameter:=CHANGE_ECAT_PREOP_AND_IS_DEPENDENT),
		(Index:=16#1A01,	SubIndex:=3,		ValueType:=TYPE_UDINT,		Access:=ACCESS_RW,	Eeprom:=EEPROM_YES,	AmpType:=BOTH_ROT_LIN,	WhenEnabled:=ENABLED_IMMEDIATELY,		SpecialParameter:=CHANGE_ECAT_PREOP_AND_IS_DEPENDENT),
		(Index:=16#1A01,	SubIndex:=4,		ValueType:=TYPE_UDINT,		Access:=ACCESS_RW,	Eeprom:=EEPROM_YES,	AmpType:=BOTH_ROT_LIN,	WhenEnabled:=ENABLED_IMMEDIATELY,		SpecialParameter:=CHANGE_ECAT_PREOP_AND_IS_DEPENDENT),
(*70*)	(Index:=16#1A01,	SubIndex:=5,		ValueType:=TYPE_UDINT,		Access:=ACCESS_RW,	Eeprom:=EEPROM_YES,	AmpType:=BOTH_ROT_LIN,	WhenEnabled:=ENABLED_IMMEDIATELY,		SpecialParameter:=CHANGE_ECAT_PREOP_AND_IS_DEPENDENT),
		(Index:=16#1A01,	SubIndex:=6,		ValueType:=TYPE_UDINT,		Access:=ACCESS_RW,	Eeprom:=EEPROM_YES,	AmpType:=BOTH_ROT_LIN,	WhenEnabled:=ENABLED_IMMEDIATELY,		SpecialParameter:=CHANGE_ECAT_PREOP_AND_IS_DEPENDENT),
		(Index:=16#1A01,	SubIndex:=7,		ValueType:=TYPE_UDINT,		Access:=ACCESS_RW,	Eeprom:=EEPROM_YES,	AmpType:=BOTH_ROT_LIN,	WhenEnabled:=ENABLED_IMMEDIATELY,		SpecialParameter:=CHANGE_ECAT_PREOP_AND_IS_DEPENDENT),
		(Index:=16#1A01,	SubIndex:=8,		ValueType:=TYPE_UDINT,		Access:=ACCESS_RW,	Eeprom:=EEPROM_YES,	AmpType:=BOTH_ROT_LIN,	WhenEnabled:=ENABLED_IMMEDIATELY,		SpecialParameter:=CHANGE_ECAT_PREOP_AND_IS_DEPENDENT),
		(Index:=16#1A02,	SubIndex:=0,		ValueType:=TYPE_USINT,		Access:=ACCESS_RW,	Eeprom:=EEPROM_YES,	AmpType:=BOTH_ROT_LIN,	WhenEnabled:=ENABLED_IMMEDIATELY,		SpecialParameter:=CHANGE_ECAT_PREOP_AND_HAS_DEPENDENT,		DependentValueUsint:=0),
		(Index:=16#1A02,	SubIndex:=1,		ValueType:=TYPE_UDINT,		Access:=ACCESS_RW,	Eeprom:=EEPROM_YES,	AmpType:=BOTH_ROT_LIN,	WhenEnabled:=ENABLED_IMMEDIATELY,		SpecialParameter:=CHANGE_ECAT_PREOP_AND_IS_DEPENDENT),
		(Index:=16#1A02,	SubIndex:=2,		ValueType:=TYPE_UDINT,		Access:=ACCESS_RW,	Eeprom:=EEPROM_YES,	AmpType:=BOTH_ROT_LIN,	WhenEnabled:=ENABLED_IMMEDIATELY,		SpecialParameter:=CHANGE_ECAT_PREOP_AND_IS_DEPENDENT),
		(Index:=16#1A02,	SubIndex:=3,		ValueType:=TYPE_UDINT,		Access:=ACCESS_RW,	Eeprom:=EEPROM_YES,	AmpType:=BOTH_ROT_LIN,	WhenEnabled:=ENABLED_IMMEDIATELY,		SpecialParameter:=CHANGE_ECAT_PREOP_AND_IS_DEPENDENT),
		(Index:=16#1A02,	SubIndex:=4,		ValueType:=TYPE_UDINT,		Access:=ACCESS_RW,	Eeprom:=EEPROM_YES,	AmpType:=BOTH_ROT_LIN,	WhenEnabled:=ENABLED_IMMEDIATELY,		SpecialParameter:=CHANGE_ECAT_PREOP_AND_IS_DEPENDENT),
		(Index:=16#1A02,	SubIndex:=5,		ValueType:=TYPE_UDINT,		Access:=ACCESS_RW,	Eeprom:=EEPROM_YES,	AmpType:=BOTH_ROT_LIN,	WhenEnabled:=ENABLED_IMMEDIATELY,		SpecialParameter:=CHANGE_ECAT_PREOP_AND_IS_DEPENDENT),
(*80*)	(Index:=16#1A02,	SubIndex:=6,		ValueType:=TYPE_UDINT,		Access:=ACCESS_RW,	Eeprom:=EEPROM_YES,	AmpType:=BOTH_ROT_LIN,	WhenEnabled:=ENABLED_IMMEDIATELY,		SpecialParameter:=CHANGE_ECAT_PREOP_AND_IS_DEPENDENT),
		(Index:=16#1A02,	SubIndex:=7,		ValueType:=TYPE_UDINT,		Access:=ACCESS_RW,	Eeprom:=EEPROM_YES,	AmpType:=BOTH_ROT_LIN,	WhenEnabled:=ENABLED_IMMEDIATELY,		SpecialParameter:=CHANGE_ECAT_PREOP_AND_IS_DEPENDENT),
		(Index:=16#1A02,	SubIndex:=8,		ValueType:=TYPE_UDINT,		Access:=ACCESS_RW,	Eeprom:=EEPROM_YES,	AmpType:=BOTH_ROT_LIN,	WhenEnabled:=ENABLED_IMMEDIATELY,		SpecialParameter:=CHANGE_ECAT_PREOP_AND_IS_DEPENDENT),
		(Index:=16#1A03,	SubIndex:=0,		ValueType:=TYPE_USINT,		Access:=ACCESS_RW,	Eeprom:=EEPROM_YES,	AmpType:=BOTH_ROT_LIN,	WhenEnabled:=ENABLED_IMMEDIATELY,		SpecialParameter:=CHANGE_ECAT_PREOP_AND_HAS_DEPENDENT,		DependentValueUsint:=0),
		(Index:=16#1A03,	SubIndex:=1,		ValueType:=TYPE_UDINT,		Access:=ACCESS_RW,	Eeprom:=EEPROM_YES,	AmpType:=BOTH_ROT_LIN,	WhenEnabled:=ENABLED_IMMEDIATELY,		SpecialParameter:=CHANGE_ECAT_PREOP_AND_IS_DEPENDENT),
		(Index:=16#1A03,	SubIndex:=2,		ValueType:=TYPE_UDINT,		Access:=ACCESS_RW,	Eeprom:=EEPROM_YES,	AmpType:=BOTH_ROT_LIN,	WhenEnabled:=ENABLED_IMMEDIATELY,		SpecialParameter:=CHANGE_ECAT_PREOP_AND_IS_DEPENDENT),
		(Index:=16#1A03,	SubIndex:=3,		ValueType:=TYPE_UDINT,		Access:=ACCESS_RW,	Eeprom:=EEPROM_YES,	AmpType:=BOTH_ROT_LIN,	WhenEnabled:=ENABLED_IMMEDIATELY,		SpecialParameter:=CHANGE_ECAT_PREOP_AND_IS_DEPENDENT),
		(Index:=16#1A03,	SubIndex:=4,		ValueType:=TYPE_UDINT,		Access:=ACCESS_RW,	Eeprom:=EEPROM_YES,	AmpType:=BOTH_ROT_LIN,	WhenEnabled:=ENABLED_IMMEDIATELY,		SpecialParameter:=CHANGE_ECAT_PREOP_AND_IS_DEPENDENT),
		(Index:=16#1A03,	SubIndex:=5,		ValueType:=TYPE_UDINT,		Access:=ACCESS_RW,	Eeprom:=EEPROM_YES,	AmpType:=BOTH_ROT_LIN,	WhenEnabled:=ENABLED_IMMEDIATELY,		SpecialParameter:=CHANGE_ECAT_PREOP_AND_IS_DEPENDENT),
		(Index:=16#1A03,	SubIndex:=6,		ValueType:=TYPE_UDINT,		Access:=ACCESS_RW,	Eeprom:=EEPROM_YES,	AmpType:=BOTH_ROT_LIN,	WhenEnabled:=ENABLED_IMMEDIATELY,		SpecialParameter:=CHANGE_ECAT_PREOP_AND_IS_DEPENDENT),
(*90*)	(Index:=16#1A03,	SubIndex:=7,		ValueType:=TYPE_UDINT,		Access:=ACCESS_RW,	Eeprom:=EEPROM_YES,	AmpType:=BOTH_ROT_LIN,	WhenEnabled:=ENABLED_IMMEDIATELY,		SpecialParameter:=CHANGE_ECAT_PREOP_AND_IS_DEPENDENT),
		(Index:=16#1A03,	SubIndex:=8,		ValueType:=TYPE_UDINT,		Access:=ACCESS_RW,	Eeprom:=EEPROM_YES,	AmpType:=BOTH_ROT_LIN,	WhenEnabled:=ENABLED_IMMEDIATELY,		SpecialParameter:=CHANGE_ECAT_PREOP_AND_IS_DEPENDENT),
		(Index:=16#1C00,	SubIndex:=0,		ValueType:=TYPE_USINT,		Access:=ACCESS_RO,		Eeprom:=EEPROM_NO,	AmpType:=BOTH_ROT_LIN,	WhenEnabled:=ENABLED_IMMEDIATELY),
		(Index:=16#1C00,	SubIndex:=1,		ValueType:=TYPE_USINT,		Access:=ACCESS_RO,		Eeprom:=EEPROM_NO,	AmpType:=BOTH_ROT_LIN,	WhenEnabled:=ENABLED_IMMEDIATELY),
		(Index:=16#1C00,	SubIndex:=2,		ValueType:=TYPE_USINT,		Access:=ACCESS_RO,		Eeprom:=EEPROM_NO,	AmpType:=BOTH_ROT_LIN,	WhenEnabled:=ENABLED_IMMEDIATELY),
		(Index:=16#1C00,	SubIndex:=3,		ValueType:=TYPE_USINT,		Access:=ACCESS_RO,		Eeprom:=EEPROM_NO,	AmpType:=BOTH_ROT_LIN,	WhenEnabled:=ENABLED_IMMEDIATELY),
		(Index:=16#1C00,	SubIndex:=4,		ValueType:=TYPE_USINT,		Access:=ACCESS_RO,		Eeprom:=EEPROM_NO,	AmpType:=BOTH_ROT_LIN,	WhenEnabled:=ENABLED_IMMEDIATELY),
		(Index:=16#1C10,	SubIndex:=0,		ValueType:=TYPE_USINT,		Access:=ACCESS_RO,		Eeprom:=EEPROM_NO,	AmpType:=BOTH_ROT_LIN,	WhenEnabled:=ENABLED_IMMEDIATELY),
		(Index:=16#1C11,	SubIndex:=0,		ValueType:=TYPE_USINT,		Access:=ACCESS_RO,		Eeprom:=EEPROM_NO,	AmpType:=BOTH_ROT_LIN,	WhenEnabled:=ENABLED_IMMEDIATELY),
		(Index:=16#1C12,	SubIndex:=0,		ValueType:=TYPE_USINT,		Access:=ACCESS_RW,	Eeprom:=EEPROM_YES,	AmpType:=BOTH_ROT_LIN,	WhenEnabled:=ENABLED_IMMEDIATELY,		SpecialParameter:=CHANGE_ECAT_PREOP_AND_HAS_DEPENDENT,		DependentValueUsint:=0), (*Can only be changed in the EtherCAT Pre-Operational State*)
(*100*)	(Index:=16#1C12,	SubIndex:=1,		ValueType:=TYPE_UINT,		Access:=ACCESS_RW,	Eeprom:=EEPROM_YES,	AmpType:=BOTH_ROT_LIN,	WhenEnabled:=ENABLED_IMMEDIATELY,		SpecialParameter:=CHANGE_ECAT_PREOP_AND_IS_DEPENDENT), (*Can only be changed in Pre-Op, and Requires subindex 0 to be 0*)
		(Index:=16#1C12,	SubIndex:=2,		ValueType:=TYPE_UINT,		Access:=ACCESS_RW,	Eeprom:=EEPROM_YES,	AmpType:=BOTH_ROT_LIN,	WhenEnabled:=ENABLED_IMMEDIATELY,		SpecialParameter:=CHANGE_ECAT_PREOP_AND_IS_DEPENDENT), (*Can only be changed in Pre-Op, and Requires subindex 0 to be 0*)
		(Index:=16#1C13,	SubIndex:=0,		ValueType:=TYPE_USINT,		Access:=ACCESS_RW,	Eeprom:=EEPROM_YES,	AmpType:=BOTH_ROT_LIN,	WhenEnabled:=ENABLED_IMMEDIATELY,		SpecialParameter:=CHANGE_ECAT_PREOP_AND_HAS_DEPENDENT,		DependentValueUsint:=0), (*Can only be changed in the EtherCAT Pre-Operational State*)
		(Index:=16#1C13,	SubIndex:=1,		ValueType:=TYPE_UINT,		Access:=ACCESS_RW,	Eeprom:=EEPROM_YES,	AmpType:=BOTH_ROT_LIN,	WhenEnabled:=ENABLED_IMMEDIATELY,		SpecialParameter:=CHANGE_ECAT_PREOP_AND_IS_DEPENDENT), (*Can only be changed in Pre-Op, and Requires subindex 0 to be 0*)
		(Index:=16#1C13,	SubIndex:=2,		ValueType:=TYPE_UINT,		Access:=ACCESS_RW,	Eeprom:=EEPROM_YES,	AmpType:=BOTH_ROT_LIN,	WhenEnabled:=ENABLED_IMMEDIATELY,		SpecialParameter:=CHANGE_ECAT_PREOP_AND_IS_DEPENDENT), (*Can only be changed in Pre-Op, and Requires subindex 0 to be 0*)
		(Index:=16#1C32,	SubIndex:=0,		ValueType:=TYPE_USINT,		Access:=ACCESS_RO,		Eeprom:=EEPROM_NO,	AmpType:=BOTH_ROT_LIN,	WhenEnabled:=ENABLED_IMMEDIATELY),
		(Index:=16#1C32,	SubIndex:=1,		ValueType:=TYPE_UINT,		Access:=ACCESS_RO,		Eeprom:=EEPROM_NO,	AmpType:=BOTH_ROT_LIN,	WhenEnabled:=ENABLED_IMMEDIATELY),
		(Index:=16#1C32,	SubIndex:=2,		ValueType:=TYPE_UDINT,		Access:=ACCESS_RO,		Eeprom:=EEPROM_NO,	AmpType:=BOTH_ROT_LIN,	WhenEnabled:=ENABLED_IMMEDIATELY),
		(Index:=16#1C32,	SubIndex:=3,		ValueType:=TYPE_UDINT,		Access:=ACCESS_RO,		Eeprom:=EEPROM_NO,	AmpType:=BOTH_ROT_LIN,	WhenEnabled:=ENABLED_IMMEDIATELY),
		(Index:=16#1C32,	SubIndex:=4,		ValueType:=TYPE_UINT,		Access:=ACCESS_RO,		Eeprom:=EEPROM_NO,	AmpType:=BOTH_ROT_LIN,	WhenEnabled:=ENABLED_IMMEDIATELY),
(*110*)	(Index:=16#1C32,	SubIndex:=5,		ValueType:=TYPE_UDINT,		Access:=ACCESS_RO,		Eeprom:=EEPROM_NO,	AmpType:=BOTH_ROT_LIN,	WhenEnabled:=ENABLED_IMMEDIATELY),
		(Index:=16#1C32,	SubIndex:=6,		ValueType:=TYPE_UDINT,		Access:=ACCESS_RO,		Eeprom:=EEPROM_NO,	AmpType:=BOTH_ROT_LIN,	WhenEnabled:=ENABLED_IMMEDIATELY),
		(Index:=16#1C32,	SubIndex:=7,		ValueType:=TYPE_UDINT,		Access:=ACCESS_RO,		Eeprom:=EEPROM_NO,	AmpType:=BOTH_ROT_LIN,	WhenEnabled:=ENABLED_IMMEDIATELY),
		(Index:=16#1C32,	SubIndex:=8,		ValueType:=TYPE_UINT,		Access:=ACCESS_RO,		Eeprom:=EEPROM_NO,	AmpType:=BOTH_ROT_LIN,	WhenEnabled:=ENABLED_IMMEDIATELY),
		(Index:=16#1C32,	SubIndex:=9,		ValueType:=TYPE_UDINT,		Access:=ACCESS_RO,		Eeprom:=EEPROM_NO,	AmpType:=BOTH_ROT_LIN,	WhenEnabled:=ENABLED_IMMEDIATELY),
		(Index:=16#1C32,	SubIndex:=10,		ValueType:=TYPE_UDINT,		Access:=ACCESS_RO,		Eeprom:=EEPROM_NO,	AmpType:=BOTH_ROT_LIN,	WhenEnabled:=ENABLED_IMMEDIATELY),
		(Index:=16#1C32,	SubIndex:=11,		ValueType:=TYPE_UDINT,		Access:=ACCESS_RO,		Eeprom:=EEPROM_NO,	AmpType:=BOTH_ROT_LIN,	WhenEnabled:=ENABLED_IMMEDIATELY),
		(Index:=16#1C32,	SubIndex:=12,		ValueType:=TYPE_UDINT,		Access:=ACCESS_RO,		Eeprom:=EEPROM_NO,	AmpType:=BOTH_ROT_LIN,	WhenEnabled:=ENABLED_IMMEDIATELY),
		(Index:=16#1C33,	SubIndex:=0,		ValueType:=TYPE_USINT,		Access:=ACCESS_RO,		Eeprom:=EEPROM_NO,	AmpType:=BOTH_ROT_LIN,	WhenEnabled:=ENABLED_IMMEDIATELY),
		(Index:=16#1C33,	SubIndex:=1,		ValueType:=TYPE_UINT,		Access:=ACCESS_RO,		Eeprom:=EEPROM_NO,	AmpType:=BOTH_ROT_LIN,	WhenEnabled:=ENABLED_IMMEDIATELY),
(*120*)	(Index:=16#1C33,	SubIndex:=2,		ValueType:=TYPE_UDINT,		Access:=ACCESS_RO,		Eeprom:=EEPROM_NO,	AmpType:=BOTH_ROT_LIN,	WhenEnabled:=ENABLED_IMMEDIATELY),
		(Index:=16#1C33,	SubIndex:=3,		ValueType:=TYPE_UDINT,		Access:=ACCESS_RW,	Eeprom:=EEPROM_YES,	AmpType:=BOTH_ROT_LIN,	WhenEnabled:=ENABLED_IMMEDIATELY),
		(Index:=16#1C33,	SubIndex:=4,		ValueType:=TYPE_UINT,		Access:=ACCESS_RO,		Eeprom:=EEPROM_NO,	AmpType:=BOTH_ROT_LIN,	WhenEnabled:=ENABLED_IMMEDIATELY),
		(Index:=16#1C33,	SubIndex:=5,		ValueType:=TYPE_UDINT,		Access:=ACCESS_RO,		Eeprom:=EEPROM_NO,	AmpType:=BOTH_ROT_LIN,	WhenEnabled:=ENABLED_IMMEDIATELY),
		(Index:=16#1C33,	SubIndex:=6,		ValueType:=TYPE_UDINT,		Access:=ACCESS_RO,		Eeprom:=EEPROM_NO,	AmpType:=BOTH_ROT_LIN,	WhenEnabled:=ENABLED_IMMEDIATELY),
		(Index:=16#1C33,	SubIndex:=7,		ValueType:=TYPE_UDINT,		Access:=ACCESS_RO,		Eeprom:=EEPROM_NO,	AmpType:=BOTH_ROT_LIN,	WhenEnabled:=ENABLED_IMMEDIATELY),
		(Index:=16#1C33,	SubIndex:=8,		ValueType:=TYPE_UINT,		Access:=ACCESS_RO,		Eeprom:=EEPROM_NO,	AmpType:=BOTH_ROT_LIN,	WhenEnabled:=ENABLED_IMMEDIATELY),
		(Index:=16#1C33,	SubIndex:=9,		ValueType:=TYPE_UDINT,		Access:=ACCESS_RO,		Eeprom:=EEPROM_NO,	AmpType:=BOTH_ROT_LIN,	WhenEnabled:=ENABLED_IMMEDIATELY),
		(Index:=16#1C33,	SubIndex:=10,		ValueType:=TYPE_UDINT,		Access:=ACCESS_RO,		Eeprom:=EEPROM_NO,	AmpType:=BOTH_ROT_LIN,	WhenEnabled:=ENABLED_IMMEDIATELY),
		(Index:=16#1F01,	SubIndex:=0,		ValueType:=TYPE_USINT,		Access:=ACCESS_RO,		Eeprom:=EEPROM_NO,	AmpType:=BOTH_ROT_LIN,	WhenEnabled:=ENABLED_IMMEDIATELY),
(*130*)	(Index:=16#1F01,	SubIndex:=1,		ValueType:=TYPE_UDINT,		Access:=ACCESS_RO,		Eeprom:=EEPROM_NO,	AmpType:=BOTH_ROT_LIN,	WhenEnabled:=ENABLED_IMMEDIATELY),
		(Index:=16#1F01,	SubIndex:=2,		ValueType:=TYPE_UDINT,		Access:=ACCESS_RW,	Eeprom:=EEPROM_NO,	AmpType:=BOTH_ROT_LIN,	WhenEnabled:=ENABLED_IMMEDIATELY),
		(Index:=16#2000,	SubIndex:=0,		ValueType:=TYPE_UINT,		Access:=ACCESS_RW,	Eeprom:=EEPROM_YES,	AmpType:=BOTH_ROT_LIN,	WhenEnabled:=ENABLED_AFTER_RESTART),
		(Index:=16#2001,	SubIndex:=0,		ValueType:=TYPE_UINT,		Access:=ACCESS_RW,	Eeprom:=EEPROM_YES,	AmpType:=BOTH_ROT_LIN,	WhenEnabled:=ENABLED_AFTER_RESTART),
		(Index:=16#2002,	SubIndex:=0,		ValueType:=TYPE_UINT,		Access:=ACCESS_RW,	Eeprom:=EEPROM_YES,	AmpType:=BOTH_ROT_LIN,	WhenEnabled:=ENABLED_AFTER_RESTART),
		(Index:=16#2006,	SubIndex:=0,		ValueType:=TYPE_UINT,		Access:=ACCESS_RW,	Eeprom:=EEPROM_YES,	AmpType:=BOTH_ROT_LIN,	WhenEnabled:=ENABLED_IMMEDIATELY),
		(Index:=16#2007,	SubIndex:=0,		ValueType:=TYPE_UINT,		Access:=ACCESS_RW,	Eeprom:=EEPROM_YES,	AmpType:=BOTH_ROT_LIN,	WhenEnabled:=ENABLED_IMMEDIATELY),
		(Index:=16#2008,	SubIndex:=0,		ValueType:=TYPE_UINT,		Access:=ACCESS_RW,	Eeprom:=EEPROM_YES,	AmpType:=BOTH_ROT_LIN,	WhenEnabled:=ENABLED_AFTER_RESTART),
		(Index:=16#2009,	SubIndex:=0,		ValueType:=TYPE_UINT,		Access:=ACCESS_RW,	Eeprom:=EEPROM_YES,	AmpType:=BOTH_ROT_LIN,	WhenEnabled:=ENABLED_AFTER_RESTART),
		(Index:=16#200B,	SubIndex:=0,		ValueType:=TYPE_UINT,		Access:=ACCESS_RW,	Eeprom:=EEPROM_YES,	AmpType:=BOTH_ROT_LIN,	WhenEnabled:=ENABLED_AFTER_RESTART),
(*140*)	(Index:=16#200C,	SubIndex:=0,		ValueType:=TYPE_UINT,		Access:=ACCESS_RW,	Eeprom:=EEPROM_YES,	AmpType:=BOTH_ROT_LIN,	WhenEnabled:=ENABLED_AFTER_RESTART),
		(Index:=16#200D,	SubIndex:=0,		ValueType:=TYPE_UINT,		Access:=ACCESS_RW,	Eeprom:=EEPROM_YES,	AmpType:=BOTH_ROT_LIN,	WhenEnabled:=ENABLED_AFTER_RESTART),
		(Index:=16#2010,	SubIndex:=0,		ValueType:=TYPE_UINT,		Access:=ACCESS_RW,	Eeprom:=EEPROM_YES,	AmpType:=BOTH_ROT_LIN,	WhenEnabled:=ENABLED_AFTER_RESTART),
		(Index:=16#2080,	SubIndex:=0,		ValueType:=TYPE_UINT,		Access:=ACCESS_RW,	Eeprom:=EEPROM_YES,	AmpType:=LINEAR,			WhenEnabled:=ENABLED_AFTER_RESTART),
		(Index:=16#2100,	SubIndex:=0,		ValueType:=TYPE_UINT,		Access:=ACCESS_RW,	Eeprom:=EEPROM_YES,	AmpType:=BOTH_ROT_LIN,	WhenEnabled:=ENABLED_IMMEDIATELY),
		(Index:=16#2101,	SubIndex:=0,		ValueType:=TYPE_UINT,		Access:=ACCESS_RW,	Eeprom:=EEPROM_YES,	AmpType:=BOTH_ROT_LIN,	WhenEnabled:=ENABLED_IMMEDIATELY),
		(Index:=16#2102,	SubIndex:=0,		ValueType:=TYPE_UINT,		Access:=ACCESS_RW,	Eeprom:=EEPROM_YES,	AmpType:=BOTH_ROT_LIN,	WhenEnabled:=ENABLED_IMMEDIATELY),
		(Index:=16#2103,	SubIndex:=0,		ValueType:=TYPE_UINT,		Access:=ACCESS_RW,	Eeprom:=EEPROM_YES,	AmpType:=BOTH_ROT_LIN,	WhenEnabled:=ENABLED_IMMEDIATELY),
		(Index:=16#2104,	SubIndex:=0,		ValueType:=TYPE_UINT,		Access:=ACCESS_RW,	Eeprom:=EEPROM_YES,	AmpType:=BOTH_ROT_LIN,	WhenEnabled:=ENABLED_IMMEDIATELY),
		(Index:=16#2105,	SubIndex:=0,		ValueType:=TYPE_UINT,		Access:=ACCESS_RW,	Eeprom:=EEPROM_YES,	AmpType:=BOTH_ROT_LIN,	WhenEnabled:=ENABLED_IMMEDIATELY),
(*150*)	(Index:=16#2106,	SubIndex:=0,		ValueType:=TYPE_UINT,		Access:=ACCESS_RW,	Eeprom:=EEPROM_YES,	AmpType:=BOTH_ROT_LIN,	WhenEnabled:=ENABLED_IMMEDIATELY),
		(Index:=16#2109,	SubIndex:=0,		ValueType:=TYPE_UINT,		Access:=ACCESS_RW,	Eeprom:=EEPROM_YES,	AmpType:=BOTH_ROT_LIN,	WhenEnabled:=ENABLED_IMMEDIATELY),
		(Index:=16#210A,	SubIndex:=0,		ValueType:=TYPE_UINT,		Access:=ACCESS_RW,	Eeprom:=EEPROM_YES,	AmpType:=BOTH_ROT_LIN,	WhenEnabled:=ENABLED_IMMEDIATELY),
		(Index:=16#210B,	SubIndex:=0,		ValueType:=TYPE_UINT,		Access:=ACCESS_RW,	Eeprom:=EEPROM_YES,	AmpType:=BOTH_ROT_LIN,	WhenEnabled:=ENABLED_SPECIAL,			EnRestartPattern:=16#0010),
		(Index:=16#210C,	SubIndex:=0,		ValueType:=TYPE_UINT,		Access:=ACCESS_RW,	Eeprom:=EEPROM_YES,	AmpType:=BOTH_ROT_LIN,	WhenEnabled:=ENABLED_IMMEDIATELY),
		(Index:=16#210D,	SubIndex:=0,		ValueType:=TYPE_UINT,		Access:=ACCESS_RW,	Eeprom:=EEPROM_YES,	AmpType:=ROTARY,			WhenEnabled:=ENABLED_IMMEDIATELY),
		(Index:=16#210E,	SubIndex:=0,		ValueType:=TYPE_UINT,		Access:=ACCESS_RW,	Eeprom:=EEPROM_YES,	AmpType:=ROTARY,			WhenEnabled:=ENABLED_IMMEDIATELY),
		(Index:=16#210F,	SubIndex:=0,		ValueType:=TYPE_UINT,		Access:=ACCESS_RW,	Eeprom:=EEPROM_YES,	AmpType:=BOTH_ROT_LIN,	WhenEnabled:=ENABLED_IMMEDIATELY),
		(Index:=16#211F,	SubIndex:=0,		ValueType:=TYPE_UINT,		Access:=ACCESS_RW,	Eeprom:=EEPROM_YES,	AmpType:=BOTH_ROT_LIN,	WhenEnabled:=ENABLED_IMMEDIATELY),
		(Index:=16#2121,	SubIndex:=0,		ValueType:=TYPE_UINT,		Access:=ACCESS_RW,	Eeprom:=EEPROM_YES,	AmpType:=BOTH_ROT_LIN,	WhenEnabled:=ENABLED_IMMEDIATELY),
(*160*)	(Index:=16#2122,	SubIndex:=0,		ValueType:=TYPE_UINT,		Access:=ACCESS_RW,	Eeprom:=EEPROM_YES,	AmpType:=BOTH_ROT_LIN,	WhenEnabled:=ENABLED_IMMEDIATELY),
		(Index:=16#2123,	SubIndex:=0,		ValueType:=TYPE_UINT,		Access:=ACCESS_RW,	Eeprom:=EEPROM_YES,	AmpType:=BOTH_ROT_LIN,	WhenEnabled:=ENABLED_IMMEDIATELY),
		(Index:=16#2124,	SubIndex:=0,		ValueType:=TYPE_UINT,		Access:=ACCESS_RW,	Eeprom:=EEPROM_YES,	AmpType:=BOTH_ROT_LIN,	WhenEnabled:=ENABLED_IMMEDIATELY),
		(Index:=16#2125,	SubIndex:=0,		ValueType:=TYPE_UINT,		Access:=ACCESS_RW,	Eeprom:=EEPROM_YES,	AmpType:=BOTH_ROT_LIN,	WhenEnabled:=ENABLED_IMMEDIATELY),
		(Index:=16#2131,	SubIndex:=0,		ValueType:=TYPE_UINT,		Access:=ACCESS_RW,	Eeprom:=EEPROM_YES,	AmpType:=BOTH_ROT_LIN,	WhenEnabled:=ENABLED_IMMEDIATELY),
		(Index:=16#2132,	SubIndex:=0,		ValueType:=TYPE_UINT,		Access:=ACCESS_RW,	Eeprom:=EEPROM_YES,	AmpType:=BOTH_ROT_LIN,	WhenEnabled:=ENABLED_IMMEDIATELY),
		(Index:=16#2135,	SubIndex:=0,		ValueType:=TYPE_UINT,		Access:=ACCESS_RW,	Eeprom:=EEPROM_YES,	AmpType:=BOTH_ROT_LIN,	WhenEnabled:=ENABLED_IMMEDIATELY),
		(Index:=16#2136,	SubIndex:=0,		ValueType:=TYPE_UINT,		Access:=ACCESS_RW,	Eeprom:=EEPROM_YES,	AmpType:=BOTH_ROT_LIN,	WhenEnabled:=ENABLED_IMMEDIATELY),
		(Index:=16#2139,	SubIndex:=0,		ValueType:=TYPE_UINT,		Access:=ACCESS_RW,	Eeprom:=EEPROM_YES,	AmpType:=BOTH_ROT_LIN,	WhenEnabled:=ENABLED_IMMEDIATELY),
		(Index:=16#213D,	SubIndex:=0,		ValueType:=TYPE_UINT,		Access:=ACCESS_RW,	Eeprom:=EEPROM_YES,	AmpType:=BOTH_ROT_LIN,	WhenEnabled:=ENABLED_IMMEDIATELY),
(*170*)	(Index:=16#2140,	SubIndex:=0,		ValueType:=TYPE_UINT,		Access:=ACCESS_RW,	Eeprom:=EEPROM_YES,	AmpType:=BOTH_ROT_LIN,	WhenEnabled:=ENABLED_IMMEDIATELY),
		(Index:=16#2141,	SubIndex:=0,		ValueType:=TYPE_UINT,		Access:=ACCESS_RW,	Eeprom:=EEPROM_YES,	AmpType:=BOTH_ROT_LIN,	WhenEnabled:=ENABLED_IMMEDIATELY),
		(Index:=16#2142,	SubIndex:=0,		ValueType:=TYPE_UINT,		Access:=ACCESS_RW,	Eeprom:=EEPROM_YES,	AmpType:=BOTH_ROT_LIN,	WhenEnabled:=ENABLED_IMMEDIATELY),
		(Index:=16#2143,	SubIndex:=0,		ValueType:=TYPE_UINT,		Access:=ACCESS_RW,	Eeprom:=EEPROM_YES,	AmpType:=BOTH_ROT_LIN,	WhenEnabled:=ENABLED_IMMEDIATELY),
		(Index:=16#2144,	SubIndex:=0,		ValueType:=TYPE_UINT,		Access:=ACCESS_RW,	Eeprom:=EEPROM_YES,	AmpType:=BOTH_ROT_LIN,	WhenEnabled:=ENABLED_IMMEDIATELY),
		(Index:=16#2145,	SubIndex:=0,		ValueType:=TYPE_UINT,		Access:=ACCESS_RW,	Eeprom:=EEPROM_YES,	AmpType:=BOTH_ROT_LIN,	WhenEnabled:=ENABLED_IMMEDIATELY),
		(Index:=16#2146,	SubIndex:=0,		ValueType:=TYPE_UINT,		Access:=ACCESS_RW,	Eeprom:=EEPROM_YES,	AmpType:=BOTH_ROT_LIN,	WhenEnabled:=ENABLED_IMMEDIATELY),
		(Index:=16#2147,	SubIndex:=0,		ValueType:=TYPE_UINT,		Access:=ACCESS_RW,	Eeprom:=EEPROM_YES,	AmpType:=BOTH_ROT_LIN,	WhenEnabled:=ENABLED_IMMEDIATELY),
		(Index:=16#2148,	SubIndex:=0,		ValueType:=TYPE_UINT,		Access:=ACCESS_RW,	Eeprom:=EEPROM_YES,	AmpType:=BOTH_ROT_LIN,	WhenEnabled:=ENABLED_IMMEDIATELY),
		(Index:=16#2149,	SubIndex:=0,		ValueType:=TYPE_UINT,		Access:=ACCESS_RW,	Eeprom:=EEPROM_YES,	AmpType:=BOTH_ROT_LIN,	WhenEnabled:=ENABLED_IMMEDIATELY),
(*180*)	(Index:=16#214A,	SubIndex:=0,		ValueType:=TYPE_UINT,		Access:=ACCESS_RW,	Eeprom:=EEPROM_YES,	AmpType:=BOTH_ROT_LIN,	WhenEnabled:=ENABLED_IMMEDIATELY),
		(Index:=16#214B,	SubIndex:=0,		ValueType:=TYPE_UINT,		Access:=ACCESS_RW,	Eeprom:=EEPROM_YES,	AmpType:=BOTH_ROT_LIN,	WhenEnabled:=ENABLED_IMMEDIATELY),
		(Index:=16#2160,	SubIndex:=0,		ValueType:=TYPE_UINT,		Access:=ACCESS_RW,	Eeprom:=EEPROM_YES,	AmpType:=BOTH_ROT_LIN,	WhenEnabled:=ENABLED_AFTER_RESTART),
		(Index:=16#2161,	SubIndex:=0,		ValueType:=TYPE_UINT,		Access:=ACCESS_RW,	Eeprom:=EEPROM_YES,	AmpType:=BOTH_ROT_LIN,	WhenEnabled:=ENABLED_IMMEDIATELY),
		(Index:=16#2162,	SubIndex:=0,		ValueType:=TYPE_UINT,		Access:=ACCESS_RW,	Eeprom:=EEPROM_YES,	AmpType:=BOTH_ROT_LIN,	WhenEnabled:=ENABLED_IMMEDIATELY),
		(Index:=16#2163,	SubIndex:=0,		ValueType:=TYPE_UINT,		Access:=ACCESS_RW,	Eeprom:=EEPROM_YES,	AmpType:=BOTH_ROT_LIN,	WhenEnabled:=ENABLED_IMMEDIATELY),
		(Index:=16#2164,	SubIndex:=0,		ValueType:=TYPE_UINT,		Access:=ACCESS_RW,	Eeprom:=EEPROM_YES,	AmpType:=BOTH_ROT_LIN,	WhenEnabled:=ENABLED_IMMEDIATELY),
		(Index:=16#2165,	SubIndex:=0,		ValueType:=TYPE_UINT,		Access:=ACCESS_RW,	Eeprom:=EEPROM_YES,	AmpType:=BOTH_ROT_LIN,	WhenEnabled:=ENABLED_IMMEDIATELY),
		(Index:=16#2170,	SubIndex:=0,		ValueType:=TYPE_UINT,		Access:=ACCESS_RW,	Eeprom:=EEPROM_YES,	AmpType:=BOTH_ROT_LIN,	WhenEnabled:=ENABLED_SPECIAL,			EnRestartPattern:=16#0011),
		(Index:=16#2181,	SubIndex:=0,		ValueType:=TYPE_UINT,		Access:=ACCESS_RW,	Eeprom:=EEPROM_YES,	AmpType:=LINEAR,			WhenEnabled:=ENABLED_IMMEDIATELY),
(*190*)	(Index:=16#2182,	SubIndex:=0,		ValueType:=TYPE_UINT,		Access:=ACCESS_RW,	Eeprom:=EEPROM_YES,	AmpType:=LINEAR,			WhenEnabled:=ENABLED_IMMEDIATELY),
		(Index:=16#2205,	SubIndex:=0,		ValueType:=TYPE_UINT,		Access:=ACCESS_RW,	Eeprom:=EEPROM_YES,	AmpType:=ROTARY,			WhenEnabled:=ENABLED_AFTER_RESTART),
		(Index:=16#2207,	SubIndex:=0,		ValueType:=TYPE_UINT,		Access:=ACCESS_RW,	Eeprom:=EEPROM_YES,	AmpType:=BOTH_ROT_LIN,	WhenEnabled:=ENABLED_AFTER_RESTART),
		(Index:=16#220A,	SubIndex:=0,		ValueType:=TYPE_UDINT,		Access:=ACCESS_RW,	Eeprom:=EEPROM_YES,	AmpType:=ROTARY,			WhenEnabled:=ENABLED_AFTER_RESTART),
		(Index:=16#220E,	SubIndex:=0,		ValueType:=TYPE_UDINT,		Access:=ACCESS_RO,		Eeprom:=EEPROM_YES,	AmpType:=BOTH_ROT_LIN,	WhenEnabled:=ENABLED_AFTER_RESTART),
		(Index:=16#2210,	SubIndex:=0,		ValueType:=TYPE_UDINT,		Access:=ACCESS_RO,		Eeprom:=EEPROM_YES,	AmpType:=BOTH_ROT_LIN,	WhenEnabled:=ENABLED_AFTER_RESTART),
		(Index:=16#2212,	SubIndex:=0,		ValueType:=TYPE_UDINT,		Access:=ACCESS_RW,	Eeprom:=EEPROM_YES,	AmpType:=ROTARY,			WhenEnabled:=ENABLED_AFTER_RESTART),
		(Index:=16#222A,	SubIndex:=0,		ValueType:=TYPE_UINT,		Access:=ACCESS_RW,	Eeprom:=EEPROM_YES,	AmpType:=BOTH_ROT_LIN,	WhenEnabled:=ENABLED_AFTER_RESTART),
		(Index:=16#2281,	SubIndex:=0,		ValueType:=TYPE_UINT,		Access:=ACCESS_RW,	Eeprom:=EEPROM_YES,	AmpType:=BOTH_ROT_LIN,	WhenEnabled:=ENABLED_AFTER_RESTART),
		(Index:=16#2282,	SubIndex:=0,		ValueType:=TYPE_UINT,		Access:=ACCESS_RW,	Eeprom:=EEPROM_YES,	AmpType:=LINEAR,			WhenEnabled:=ENABLED_AFTER_RESTART),
(*200*)	(Index:=16#2304,	SubIndex:=0,		ValueType:=TYPE_UINT,		Access:=ACCESS_RW,	Eeprom:=EEPROM_YES,	AmpType:=ROTARY,			WhenEnabled:=ENABLED_IMMEDIATELY),
		(Index:=16#2305,	SubIndex:=0,		ValueType:=TYPE_UINT,		Access:=ACCESS_RW,	Eeprom:=EEPROM_YES,	AmpType:=BOTH_ROT_LIN,	WhenEnabled:=ENABLED_IMMEDIATELY),
		(Index:=16#2306,	SubIndex:=0,		ValueType:=TYPE_UINT,		Access:=ACCESS_RW,	Eeprom:=EEPROM_YES,	AmpType:=BOTH_ROT_LIN,	WhenEnabled:=ENABLED_IMMEDIATELY),
		(Index:=16#2310,	SubIndex:=0,		ValueType:=TYPE_UINT,		Access:=ACCESS_RW,	Eeprom:=EEPROM_YES,	AmpType:=BOTH_ROT_LIN,	WhenEnabled:=ENABLED_IMMEDIATELY),
		(Index:=16#2311,	SubIndex:=0,		ValueType:=TYPE_UINT,		Access:=ACCESS_RW,	Eeprom:=EEPROM_YES,	AmpType:=BOTH_ROT_LIN,	WhenEnabled:=ENABLED_IMMEDIATELY),
		(Index:=16#2312,	SubIndex:=0,		ValueType:=TYPE_UINT,		Access:=ACCESS_RW,	Eeprom:=EEPROM_YES,	AmpType:=ROTARY,			WhenEnabled:=ENABLED_IMMEDIATELY),
		(Index:=16#2324,	SubIndex:=0,		ValueType:=TYPE_UINT,		Access:=ACCESS_RW,	Eeprom:=EEPROM_YES,	AmpType:=BOTH_ROT_LIN,	WhenEnabled:=ENABLED_IMMEDIATELY),
		(Index:=16#2383,	SubIndex:=0,		ValueType:=TYPE_UINT,		Access:=ACCESS_RW,	Eeprom:=EEPROM_YES,	AmpType:=LINEAR,			WhenEnabled:=ENABLED_IMMEDIATELY),
		(Index:=16#2384,	SubIndex:=0,		ValueType:=TYPE_UINT,		Access:=ACCESS_RW,	Eeprom:=EEPROM_YES,	AmpType:=LINEAR,			WhenEnabled:=ENABLED_IMMEDIATELY),
		(Index:=16#2385,	SubIndex:=0,		ValueType:=TYPE_UINT,		Access:=ACCESS_RW,	Eeprom:=EEPROM_YES,	AmpType:=LINEAR,			WhenEnabled:=ENABLED_AFTER_RESTART),
(*210*)	(Index:=16#2401,	SubIndex:=0,		ValueType:=TYPE_UINT,		Access:=ACCESS_RW,	Eeprom:=EEPROM_YES,	AmpType:=BOTH_ROT_LIN,	WhenEnabled:=ENABLED_IMMEDIATELY),
		(Index:=16#2402,	SubIndex:=0,		ValueType:=TYPE_UINT,		Access:=ACCESS_RW,	Eeprom:=EEPROM_YES,	AmpType:=ROTARY,			WhenEnabled:=ENABLED_IMMEDIATELY),
		(Index:=16#2403,	SubIndex:=0,		ValueType:=TYPE_UINT,		Access:=ACCESS_RW,	Eeprom:=EEPROM_YES,	AmpType:=ROTARY,			WhenEnabled:=ENABLED_IMMEDIATELY),
		(Index:=16#2404,	SubIndex:=0,		ValueType:=TYPE_UINT,		Access:=ACCESS_RW,	Eeprom:=EEPROM_YES,	AmpType:=BOTH_ROT_LIN,	WhenEnabled:=ENABLED_IMMEDIATELY),
		(Index:=16#2405,	SubIndex:=0,		ValueType:=TYPE_UINT,		Access:=ACCESS_RW,	Eeprom:=EEPROM_YES,	AmpType:=BOTH_ROT_LIN,	WhenEnabled:=ENABLED_IMMEDIATELY),
		(Index:=16#2406,	SubIndex:=0,		ValueType:=TYPE_UINT,		Access:=ACCESS_RW,	Eeprom:=EEPROM_YES,	AmpType:=BOTH_ROT_LIN,	WhenEnabled:=ENABLED_IMMEDIATELY),
		(Index:=16#2407,	SubIndex:=0,		ValueType:=TYPE_UINT,		Access:=ACCESS_RW,	Eeprom:=EEPROM_YES,	AmpType:=ROTARY,			WhenEnabled:=ENABLED_IMMEDIATELY),
		(Index:=16#2408,	SubIndex:=0,		ValueType:=TYPE_UINT,		Access:=ACCESS_RW,	Eeprom:=EEPROM_YES,	AmpType:=BOTH_ROT_LIN,	WhenEnabled:=ENABLED_SPECIAL,			EnRestartPattern:=16#0010),
		(Index:=16#2409,	SubIndex:=0,		ValueType:=TYPE_UINT,		Access:=ACCESS_RW,	Eeprom:=EEPROM_YES,	AmpType:=BOTH_ROT_LIN,	WhenEnabled:=ENABLED_IMMEDIATELY),
		(Index:=16#240A,	SubIndex:=0,		ValueType:=TYPE_UINT,		Access:=ACCESS_RW,	Eeprom:=EEPROM_YES,	AmpType:=BOTH_ROT_LIN,	WhenEnabled:=ENABLED_IMMEDIATELY),
(*220*)	(Index:=16#240B,	SubIndex:=0,		ValueType:=TYPE_UINT,		Access:=ACCESS_RW,	Eeprom:=EEPROM_YES,	AmpType:=BOTH_ROT_LIN,	WhenEnabled:=ENABLED_IMMEDIATELY),
		(Index:=16#240C,	SubIndex:=0,		ValueType:=TYPE_UINT,		Access:=ACCESS_RW,	Eeprom:=EEPROM_YES,	AmpType:=BOTH_ROT_LIN,	WhenEnabled:=ENABLED_IMMEDIATELY),
		(Index:=16#240D,	SubIndex:=0,		ValueType:=TYPE_UINT,		Access:=ACCESS_RW,	Eeprom:=EEPROM_YES,	AmpType:=BOTH_ROT_LIN,	WhenEnabled:=ENABLED_IMMEDIATELY),
		(Index:=16#240E,	SubIndex:=0,		ValueType:=TYPE_UINT,		Access:=ACCESS_RW,	Eeprom:=EEPROM_YES,	AmpType:=BOTH_ROT_LIN,	WhenEnabled:=ENABLED_IMMEDIATELY),
		(Index:=16#240F,	SubIndex:=0,		ValueType:=TYPE_UINT,		Access:=ACCESS_RW,	Eeprom:=EEPROM_YES,	AmpType:=BOTH_ROT_LIN,	WhenEnabled:=ENABLED_IMMEDIATELY),
		(Index:=16#2410,	SubIndex:=0,		ValueType:=TYPE_UINT,		Access:=ACCESS_RW,	Eeprom:=EEPROM_YES,	AmpType:=BOTH_ROT_LIN,	WhenEnabled:=ENABLED_IMMEDIATELY),
		(Index:=16#2412,	SubIndex:=0,		ValueType:=TYPE_UINT,		Access:=ACCESS_RW,	Eeprom:=EEPROM_YES,	AmpType:=BOTH_ROT_LIN,	WhenEnabled:=ENABLED_IMMEDIATELY),
		(Index:=16#2424,	SubIndex:=0,		ValueType:=TYPE_UINT,		Access:=ACCESS_RW,	Eeprom:=EEPROM_YES,	AmpType:=BOTH_ROT_LIN,	WhenEnabled:=ENABLED_IMMEDIATELY),
		(Index:=16#2425,	SubIndex:=0,		ValueType:=TYPE_UINT,		Access:=ACCESS_RW,	Eeprom:=EEPROM_YES,	AmpType:=BOTH_ROT_LIN,	WhenEnabled:=ENABLED_IMMEDIATELY),
		(Index:=16#2456,	SubIndex:=0,		ValueType:=TYPE_UINT,		Access:=ACCESS_RW,	Eeprom:=EEPROM_YES,	AmpType:=BOTH_ROT_LIN,	WhenEnabled:=ENABLED_IMMEDIATELY),
(*230*)	(Index:=16#2460,	SubIndex:=0,		ValueType:=TYPE_UINT,		Access:=ACCESS_RW,	Eeprom:=EEPROM_YES,	AmpType:=BOTH_ROT_LIN,	WhenEnabled:=ENABLED_IMMEDIATELY),
		(Index:=16#2480,	SubIndex:=0,		ValueType:=TYPE_UINT,		Access:=ACCESS_RW,	Eeprom:=EEPROM_YES,	AmpType:=LINEAR,			WhenEnabled:=ENABLED_IMMEDIATELY),
		(Index:=16#2481,	SubIndex:=0,		ValueType:=TYPE_UINT,		Access:=ACCESS_RW,	Eeprom:=EEPROM_YES,	AmpType:=LINEAR,			WhenEnabled:=ENABLED_IMMEDIATELY),
		(Index:=16#2482,	SubIndex:=0,		ValueType:=TYPE_UINT,		Access:=ACCESS_RW,	Eeprom:=EEPROM_YES,	AmpType:=LINEAR,			WhenEnabled:=ENABLED_IMMEDIATELY),
		(Index:=16#2483,	SubIndex:=0,		ValueType:=TYPE_UINT,		Access:=ACCESS_RW,	Eeprom:=EEPROM_YES,	AmpType:=LINEAR,			WhenEnabled:=ENABLED_IMMEDIATELY),
		(Index:=16#2484,	SubIndex:=0,		ValueType:=TYPE_UINT,		Access:=ACCESS_RW,	Eeprom:=EEPROM_YES,	AmpType:=LINEAR,			WhenEnabled:=ENABLED_IMMEDIATELY),
		(Index:=16#2485,	SubIndex:=0,		ValueType:=TYPE_UINT,		Access:=ACCESS_RW,	Eeprom:=EEPROM_YES,	AmpType:=LINEAR,			WhenEnabled:=ENABLED_IMMEDIATELY),
		(Index:=16#2486,	SubIndex:=0,		ValueType:=TYPE_UINT,		Access:=ACCESS_RW,	Eeprom:=EEPROM_YES,	AmpType:=LINEAR,			WhenEnabled:=ENABLED_IMMEDIATELY),
		(Index:=16#2487,	SubIndex:=0,		ValueType:=TYPE_UINT,		Access:=ACCESS_RW,	Eeprom:=EEPROM_YES,	AmpType:=LINEAR,			WhenEnabled:=ENABLED_IMMEDIATELY),
		(Index:=16#2488,	SubIndex:=0,		ValueType:=TYPE_UINT,		Access:=ACCESS_RW,	Eeprom:=EEPROM_YES,	AmpType:=LINEAR,			WhenEnabled:=ENABLED_IMMEDIATELY),
(*240*)	(Index:=16#248E,	SubIndex:=0,		ValueType:=TYPE_UINT,		Access:=ACCESS_RW,	Eeprom:=EEPROM_YES,	AmpType:=LINEAR,			WhenEnabled:=ENABLED_IMMEDIATELY),
		(Index:=16#2490,	SubIndex:=0,		ValueType:=TYPE_UINT,		Access:=ACCESS_RW,	Eeprom:=EEPROM_YES,	AmpType:=LINEAR,			WhenEnabled:=ENABLED_IMMEDIATELY),
		(Index:=16#2495,	SubIndex:=0,		ValueType:=TYPE_UINT,		Access:=ACCESS_RW,	Eeprom:=EEPROM_YES,	AmpType:=LINEAR,			WhenEnabled:=ENABLED_IMMEDIATELY),
		(Index:=16#2498,	SubIndex:=0,		ValueType:=TYPE_UINT,		Access:=ACCESS_RW,	Eeprom:=EEPROM_YES,	AmpType:=LINEAR,			WhenEnabled:=ENABLED_IMMEDIATELY),
		(Index:=16#2502,	SubIndex:=0,		ValueType:=TYPE_UINT,		Access:=ACCESS_RW,	Eeprom:=EEPROM_YES,	AmpType:=ROTARY,			WhenEnabled:=ENABLED_IMMEDIATELY),
		(Index:=16#2503,	SubIndex:=0,		ValueType:=TYPE_UINT,		Access:=ACCESS_RW,	Eeprom:=EEPROM_YES,	AmpType:=ROTARY,			WhenEnabled:=ENABLED_IMMEDIATELY),
		(Index:=16#2506,	SubIndex:=0,		ValueType:=TYPE_UINT,		Access:=ACCESS_RW,	Eeprom:=EEPROM_YES,	AmpType:=BOTH_ROT_LIN,	WhenEnabled:=ENABLED_IMMEDIATELY),
		(Index:=16#2507,	SubIndex:=0,		ValueType:=TYPE_UINT,		Access:=ACCESS_RW,	Eeprom:=EEPROM_YES,	AmpType:=ROTARY,			WhenEnabled:=ENABLED_IMMEDIATELY),
		(Index:=16#2508,	SubIndex:=0,		ValueType:=TYPE_UINT,		Access:=ACCESS_RW,	Eeprom:=EEPROM_YES,	AmpType:=BOTH_ROT_LIN,	WhenEnabled:=ENABLED_IMMEDIATELY),
		(Index:=16#2509,	SubIndex:=0,		ValueType:=TYPE_UINT,		Access:=ACCESS_RW,	Eeprom:=EEPROM_YES,	AmpType:=BOTH_ROT_LIN,	WhenEnabled:=ENABLED_IMMEDIATELY),
(*250*)	(Index:=16#250A,	SubIndex:=0,		ValueType:=TYPE_UINT,		Access:=ACCESS_RW,	Eeprom:=EEPROM_YES,	AmpType:=BOTH_ROT_LIN,	WhenEnabled:=ENABLED_AFTER_RESTART),
		(Index:=16#250B,	SubIndex:=0,		ValueType:=TYPE_UINT,		Access:=ACCESS_RW,	Eeprom:=EEPROM_YES,	AmpType:=BOTH_ROT_LIN,	WhenEnabled:=ENABLED_AFTER_RESTART),
		(Index:=16#250E,	SubIndex:=0,		ValueType:=TYPE_UINT,		Access:=ACCESS_RW,	Eeprom:=EEPROM_YES,	AmpType:=BOTH_ROT_LIN,	WhenEnabled:=ENABLED_AFTER_RESTART),
		(Index:=16#250F,	SubIndex:=0,		ValueType:=TYPE_UINT,		Access:=ACCESS_RW,	Eeprom:=EEPROM_YES,	AmpType:=BOTH_ROT_LIN,	WhenEnabled:=ENABLED_AFTER_RESTART),
		(Index:=16#2510,	SubIndex:=0,		ValueType:=TYPE_UINT,		Access:=ACCESS_RW,	Eeprom:=EEPROM_YES,	AmpType:=BOTH_ROT_LIN,	WhenEnabled:=ENABLED_AFTER_RESTART),
		(Index:=16#2511,	SubIndex:=0,		ValueType:=TYPE_UINT,		Access:=ACCESS_RW,	Eeprom:=EEPROM_YES,	AmpType:=BOTH_ROT_LIN,	WhenEnabled:=ENABLED_AFTER_RESTART),
		(Index:=16#2512,	SubIndex:=0,		ValueType:=TYPE_UINT,		Access:=ACCESS_RW,	Eeprom:=EEPROM_YES,	AmpType:=BOTH_ROT_LIN,	WhenEnabled:=ENABLED_AFTER_RESTART),
		(Index:=16#251B,	SubIndex:=0,		ValueType:=TYPE_UDINT,		Access:=ACCESS_RW,	Eeprom:=EEPROM_YES,	AmpType:=ROTARY,			WhenEnabled:=ENABLED_IMMEDIATELY),
		(Index:=16#251E,	SubIndex:=0,		ValueType:=TYPE_UINT,		Access:=ACCESS_RW,	Eeprom:=EEPROM_YES,	AmpType:=BOTH_ROT_LIN,	WhenEnabled:=ENABLED_IMMEDIATELY),
		(Index:=16#2520,	SubIndex:=0,		ValueType:=TYPE_UDINT,		Access:=ACCESS_RW,	Eeprom:=EEPROM_YES,	AmpType:=BOTH_ROT_LIN,	WhenEnabled:=ENABLED_IMMEDIATELY),
(*260*)	(Index:=16#2522,	SubIndex:=0,		ValueType:=TYPE_UDINT,		Access:=ACCESS_RW,	Eeprom:=EEPROM_YES,	AmpType:=BOTH_ROT_LIN,	WhenEnabled:=ENABLED_IMMEDIATELY),
		(Index:=16#2524,	SubIndex:=0,		ValueType:=TYPE_UDINT,		Access:=ACCESS_RW,	Eeprom:=EEPROM_YES,	AmpType:=BOTH_ROT_LIN,	WhenEnabled:=ENABLED_IMMEDIATELY),
		(Index:=16#2526,	SubIndex:=0,		ValueType:=TYPE_UDINT,		Access:=ACCESS_RW,	Eeprom:=EEPROM_YES,	AmpType:=BOTH_ROT_LIN,	WhenEnabled:=ENABLED_IMMEDIATELY),
		(Index:=16#2528,	SubIndex:=0,		ValueType:=TYPE_UINT,		Access:=ACCESS_RW,	Eeprom:=EEPROM_YES,	AmpType:=BOTH_ROT_LIN,	WhenEnabled:=ENABLED_IMMEDIATELY),
		(Index:=16#2529,	SubIndex:=0,		ValueType:=TYPE_UINT,		Access:=ACCESS_RW,	Eeprom:=EEPROM_YES,	AmpType:=BOTH_ROT_LIN,	WhenEnabled:=ENABLED_IMMEDIATELY),
		(Index:=16#252A,	SubIndex:=0,		ValueType:=TYPE_UINT,		Access:=ACCESS_RW,	Eeprom:=EEPROM_YES,	AmpType:=ROTARY,			WhenEnabled:=ENABLED_IMMEDIATELY),
		(Index:=16#252B,	SubIndex:=0,		ValueType:=TYPE_UINT,		Access:=ACCESS_RW,	Eeprom:=EEPROM_YES,	AmpType:=BOTH_ROT_LIN,	WhenEnabled:=ENABLED_IMMEDIATELY),
		(Index:=16#252C,	SubIndex:=0,		ValueType:=TYPE_UINT,		Access:=ACCESS_RW,	Eeprom:=EEPROM_YES,	AmpType:=BOTH_ROT_LIN,	WhenEnabled:=ENABLED_AFTER_RESTART),
		(Index:=16#2530,	SubIndex:=0,		ValueType:=TYPE_UINT,		Access:=ACCESS_RW,	Eeprom:=EEPROM_YES,	AmpType:=BOTH_ROT_LIN,	WhenEnabled:=ENABLED_IMMEDIATELY),
		(Index:=16#2531,	SubIndex:=0,		ValueType:=TYPE_UDINT,		Access:=ACCESS_RW,	Eeprom:=EEPROM_YES,	AmpType:=BOTH_ROT_LIN,	WhenEnabled:=ENABLED_IMMEDIATELY),
(*270*)	(Index:=16#2533,	SubIndex:=0,		ValueType:=TYPE_UINT,		Access:=ACCESS_RW,	Eeprom:=EEPROM_YES,	AmpType:=ROTARY,			WhenEnabled:=ENABLED_IMMEDIATELY),
		(Index:=16#2534,	SubIndex:=0,		ValueType:=TYPE_UINT,		Access:=ACCESS_RW,	Eeprom:=EEPROM_YES,	AmpType:=BOTH_ROT_LIN,	WhenEnabled:=ENABLED_IMMEDIATELY),
		(Index:=16#2535,	SubIndex:=0,		ValueType:=TYPE_UINT,		Access:=ACCESS_RW,	Eeprom:=EEPROM_YES,	AmpType:=BOTH_ROT_LIN,	WhenEnabled:=ENABLED_IMMEDIATELY),
		(Index:=16#2536,	SubIndex:=0,		ValueType:=TYPE_UINT,		Access:=ACCESS_RW,	Eeprom:=EEPROM_YES,	AmpType:=BOTH_ROT_LIN,	WhenEnabled:=ENABLED_IMMEDIATELY),
		(Index:=16#2550,	SubIndex:=0,		ValueType:=TYPE_UINT,		Access:=ACCESS_RW,	Eeprom:=EEPROM_YES,	AmpType:=BOTH_ROT_LIN,	WhenEnabled:=ENABLED_IMMEDIATELY),
		(Index:=16#2551,	SubIndex:=0,		ValueType:=TYPE_UINT,		Access:=ACCESS_RW,	Eeprom:=EEPROM_YES,	AmpType:=BOTH_ROT_LIN,	WhenEnabled:=ENABLED_IMMEDIATELY),
		(Index:=16#2552,	SubIndex:=0,		ValueType:=TYPE_UINT,		Access:=ACCESS_RW,	Eeprom:=EEPROM_YES,	AmpType:=BOTH_ROT_LIN,	WhenEnabled:=ENABLED_IMMEDIATELY),
		(Index:=16#2553,	SubIndex:=0,		ValueType:=TYPE_UINT,		Access:=ACCESS_RW,	Eeprom:=EEPROM_YES,	AmpType:=BOTH_ROT_LIN,	WhenEnabled:=ENABLED_IMMEDIATELY),
		(Index:=16#2560,	SubIndex:=0,		ValueType:=TYPE_UINT,		Access:=ACCESS_RW,	Eeprom:=EEPROM_YES,	AmpType:=BOTH_ROT_LIN,	WhenEnabled:=ENABLED_IMMEDIATELY),
		(Index:=16#2561,	SubIndex:=0,		ValueType:=TYPE_UINT,		Access:=ACCESS_RW,	Eeprom:=EEPROM_YES,	AmpType:=BOTH_ROT_LIN,	WhenEnabled:=ENABLED_IMMEDIATELY),
(*280*)	(Index:=16#2582,	SubIndex:=0,		ValueType:=TYPE_UINT,		Access:=ACCESS_RW,	Eeprom:=EEPROM_YES,	AmpType:=LINEAR,			WhenEnabled:=ENABLED_IMMEDIATELY),
		(Index:=16#2583,	SubIndex:=0,		ValueType:=TYPE_UINT,		Access:=ACCESS_RW,	Eeprom:=EEPROM_YES,	AmpType:=LINEAR,			WhenEnabled:=ENABLED_IMMEDIATELY),
		(Index:=16#2584,	SubIndex:=0,		ValueType:=TYPE_UINT,		Access:=ACCESS_RW,	Eeprom:=EEPROM_YES,	AmpType:=LINEAR,			WhenEnabled:=ENABLED_IMMEDIATELY),
		(Index:=16#2585,	SubIndex:=0,		ValueType:=TYPE_UINT,		Access:=ACCESS_RW,	Eeprom:=EEPROM_YES,	AmpType:=LINEAR,			WhenEnabled:=ENABLED_IMMEDIATELY),
		(Index:=16#2586,	SubIndex:=0,		ValueType:=TYPE_UINT,		Access:=ACCESS_RW,	Eeprom:=EEPROM_YES,	AmpType:=LINEAR,			WhenEnabled:=ENABLED_IMMEDIATELY),
		(Index:=16#2587,	SubIndex:=0,		ValueType:=TYPE_UINT,		Access:=ACCESS_RW,	Eeprom:=EEPROM_NO,	AmpType:=LINEAR,			WhenEnabled:=ENABLED_IMMEDIATELY),
		(Index:=16#2600,	SubIndex:=0,		ValueType:=TYPE_UINT,		Access:=ACCESS_RW,	Eeprom:=EEPROM_YES,	AmpType:=BOTH_ROT_LIN,	WhenEnabled:=ENABLED_IMMEDIATELY),
		(Index:=16#2700,	SubIndex:=0,		ValueType:=TYPE_UDINT,		Access:=ACCESS_RW,	Eeprom:=EEPROM_NO,	AmpType:=BOTH_ROT_LIN,	WhenEnabled:=ENABLED_IMMEDIATELY,		SpecialParameter:=OBJECT_COMMAND),
		(Index:=16#2701,	SubIndex:=0,		ValueType:=TYPE_USINT,		Access:=ACCESS_RO,		Eeprom:=EEPROM_NO,	AmpType:=BOTH_ROT_LIN,	WhenEnabled:=ENABLED_IMMEDIATELY),
		(Index:=16#2701,	SubIndex:=1,		ValueType:=TYPE_UDINT,		Access:=ACCESS_RW,	Eeprom:=EEPROM_YES,	AmpType:=BOTH_ROT_LIN,	WhenEnabled:=ENABLED_IMMEDIATELY),
(*290*)	(Index:=16#2701,	SubIndex:=2,		ValueType:=TYPE_UDINT,		Access:=ACCESS_RW,	Eeprom:=EEPROM_YES,	AmpType:=BOTH_ROT_LIN,	WhenEnabled:=ENABLED_IMMEDIATELY),
		(Index:=16#2702,	SubIndex:=0,		ValueType:=TYPE_USINT,		Access:=ACCESS_RO,		Eeprom:=EEPROM_NO,	AmpType:=BOTH_ROT_LIN,	WhenEnabled:=ENABLED_IMMEDIATELY),
		(Index:=16#2702,	SubIndex:=1,		ValueType:=TYPE_UDINT,		Access:=ACCESS_RW,	Eeprom:=EEPROM_YES,	AmpType:=BOTH_ROT_LIN,	WhenEnabled:=ENABLED_IMMEDIATELY),
		(Index:=16#2702,	SubIndex:=2,		ValueType:=TYPE_UDINT,		Access:=ACCESS_RW,	Eeprom:=EEPROM_YES,	AmpType:=BOTH_ROT_LIN,	WhenEnabled:=ENABLED_IMMEDIATELY),
		(Index:=16#2703,	SubIndex:=0,		ValueType:=TYPE_USINT,		Access:=ACCESS_RO,		Eeprom:=EEPROM_NO,	AmpType:=BOTH_ROT_LIN,	WhenEnabled:=ENABLED_IMMEDIATELY),
		(Index:=16#2703,	SubIndex:=1,		ValueType:=TYPE_UDINT,		Access:=ACCESS_RW,	Eeprom:=EEPROM_YES,	AmpType:=BOTH_ROT_LIN,	WhenEnabled:=ENABLED_IMMEDIATELY),
		(Index:=16#2703,	SubIndex:=2,		ValueType:=TYPE_UDINT,		Access:=ACCESS_RW,	Eeprom:=EEPROM_YES,	AmpType:=BOTH_ROT_LIN,	WhenEnabled:=ENABLED_IMMEDIATELY),
		(Index:=16#2710,	SubIndex:=0,		ValueType:=TYPE_USINT,		Access:=ACCESS_RO,		Eeprom:=EEPROM_NO,	AmpType:=BOTH_ROT_LIN,	WhenEnabled:=ENABLED_IMMEDIATELY,		SpecialParameter:=OBJECT_COMMAND),
		(Index:=16#2710,	SubIndex:=1,		ValueType:=TYPE_STRING,	Access:=ACCESS_RW,	Eeprom:=EEPROM_NO,	AmpType:=BOTH_ROT_LIN,	WhenEnabled:=ENABLED_IMMEDIATELY,		SpecialParameter:=OBJECT_COMMAND),
		(Index:=16#2710,	SubIndex:=2,		ValueType:=TYPE_USINT,		Access:=ACCESS_RO,		Eeprom:=EEPROM_NO,	AmpType:=BOTH_ROT_LIN,	WhenEnabled:=ENABLED_IMMEDIATELY,		SpecialParameter:=OBJECT_COMMAND),
(*300*)	(Index:=16#2710,	SubIndex:=3,		ValueType:=TYPE_STRING,	Access:=ACCESS_RO,		Eeprom:=EEPROM_NO,	AmpType:=BOTH_ROT_LIN,	WhenEnabled:=ENABLED_IMMEDIATELY,		SpecialParameter:=OBJECT_COMMAND),
		(Index:=16#27E0,	SubIndex:=0,		ValueType:=TYPE_UINT,		Access:=ACCESS_RW,	Eeprom:=EEPROM_NO,	AmpType:=BOTH_ROT_LIN,	WhenEnabled:=ENABLED_IMMEDIATELY),		(*UNDEFINED_SUBINDEX in manual*)
		(Index:=16#603F,	SubIndex:=0,		ValueType:=TYPE_UINT,		Access:=ACCESS_RO,		Eeprom:=EEPROM_NO,	AmpType:=BOTH_ROT_LIN,	WhenEnabled:=ENABLED_IMMEDIATELY),
		(Index:=16#6040,	SubIndex:=0,		ValueType:=TYPE_UINT,		Access:=ACCESS_RW,	Eeprom:=EEPROM_NO,	AmpType:=BOTH_ROT_LIN,	WhenEnabled:=ENABLED_IMMEDIATELY,		SpecialParameter:=OBJECT_COMMAND),
		(Index:=16#6041,	SubIndex:=0,		ValueType:=TYPE_UINT,		Access:=ACCESS_RO,		Eeprom:=EEPROM_NO,	AmpType:=BOTH_ROT_LIN,	WhenEnabled:=ENABLED_IMMEDIATELY),
		(Index:=16#605A,	SubIndex:=0,		ValueType:=TYPE_INT,		Access:=ACCESS_RW,	Eeprom:=EEPROM_YES,	AmpType:=BOTH_ROT_LIN,	WhenEnabled:=ENABLED_IMMEDIATELY),
		(Index:=16#605B,	SubIndex:=0,		ValueType:=TYPE_INT,		Access:=ACCESS_RW,	Eeprom:=EEPROM_YES,	AmpType:=BOTH_ROT_LIN,	WhenEnabled:=ENABLED_IMMEDIATELY),
		(Index:=16#605C,	SubIndex:=0,		ValueType:=TYPE_INT,		Access:=ACCESS_RW,	Eeprom:=EEPROM_YES,	AmpType:=BOTH_ROT_LIN,	WhenEnabled:=ENABLED_IMMEDIATELY),
		(Index:=16#605D,	SubIndex:=0,		ValueType:=TYPE_INT,		Access:=ACCESS_RW,	Eeprom:=EEPROM_YES,	AmpType:=BOTH_ROT_LIN,	WhenEnabled:=ENABLED_IMMEDIATELY),
		(Index:=16#605E,	SubIndex:=0,		ValueType:=TYPE_INT,		Access:=ACCESS_RW,	Eeprom:=EEPROM_YES,	AmpType:=BOTH_ROT_LIN,	WhenEnabled:=ENABLED_IMMEDIATELY),
(*310*)	(Index:=16#6060,	SubIndex:=0,		ValueType:=TYPE_SINT,		Access:=ACCESS_RW,	Eeprom:=EEPROM_YES,	AmpType:=BOTH_ROT_LIN,	WhenEnabled:=ENABLED_IMMEDIATELY),
		(Index:=16#6061,	SubIndex:=0,		ValueType:=TYPE_SINT,		Access:=ACCESS_RO,		Eeprom:=EEPROM_NO,	AmpType:=BOTH_ROT_LIN,	WhenEnabled:=ENABLED_IMMEDIATELY),
		(Index:=16#6062,	SubIndex:=0,		ValueType:=TYPE_DINT,		Access:=ACCESS_RO,		Eeprom:=EEPROM_NO,	AmpType:=BOTH_ROT_LIN,	WhenEnabled:=ENABLED_IMMEDIATELY),
		(Index:=16#6063,	SubIndex:=0,		ValueType:=TYPE_DINT,		Access:=ACCESS_RO,		Eeprom:=EEPROM_NO,	AmpType:=BOTH_ROT_LIN,	WhenEnabled:=ENABLED_IMMEDIATELY),
		(Index:=16#6064,	SubIndex:=0,		ValueType:=TYPE_DINT,		Access:=ACCESS_RO,		Eeprom:=EEPROM_NO,	AmpType:=BOTH_ROT_LIN,	WhenEnabled:=ENABLED_IMMEDIATELY),
		(Index:=16#6065,	SubIndex:=0,		ValueType:=TYPE_UDINT,		Access:=ACCESS_RW,	Eeprom:=EEPROM_YES,	AmpType:=BOTH_ROT_LIN,	WhenEnabled:=ENABLED_IMMEDIATELY),
		(Index:=16#6066,	SubIndex:=0,		ValueType:=TYPE_UINT,		Access:=ACCESS_RW,	Eeprom:=EEPROM_YES,	AmpType:=BOTH_ROT_LIN,	WhenEnabled:=ENABLED_IMMEDIATELY),
		(Index:=16#6067,	SubIndex:=0,		ValueType:=TYPE_UDINT,		Access:=ACCESS_RW,	Eeprom:=EEPROM_YES,	AmpType:=BOTH_ROT_LIN,	WhenEnabled:=ENABLED_IMMEDIATELY),
		(Index:=16#6068,	SubIndex:=0,		ValueType:=TYPE_UINT,		Access:=ACCESS_RW,	Eeprom:=EEPROM_YES,	AmpType:=BOTH_ROT_LIN,	WhenEnabled:=ENABLED_IMMEDIATELY),
		(Index:=16#606B,	SubIndex:=0,		ValueType:=TYPE_DINT,		Access:=ACCESS_RO,		Eeprom:=EEPROM_NO,	AmpType:=BOTH_ROT_LIN,	WhenEnabled:=ENABLED_IMMEDIATELY),
(*320*)	(Index:=16#606C,	SubIndex:=0,		ValueType:=TYPE_DINT,		Access:=ACCESS_RO,		Eeprom:=EEPROM_NO,	AmpType:=BOTH_ROT_LIN,	WhenEnabled:=ENABLED_IMMEDIATELY),
		(Index:=16#606D,	SubIndex:=0,		ValueType:=TYPE_UINT,		Access:=ACCESS_RW,	Eeprom:=EEPROM_YES,	AmpType:=BOTH_ROT_LIN,	WhenEnabled:=ENABLED_IMMEDIATELY),
		(Index:=16#606E,	SubIndex:=0,		ValueType:=TYPE_UINT,		Access:=ACCESS_RW,	Eeprom:=EEPROM_YES,	AmpType:=BOTH_ROT_LIN,	WhenEnabled:=ENABLED_IMMEDIATELY),
		(Index:=16#6071,	SubIndex:=0,		ValueType:=TYPE_INT,		Access:=ACCESS_RW,	Eeprom:=EEPROM_NO,	AmpType:=BOTH_ROT_LIN,	WhenEnabled:=ENABLED_IMMEDIATELY),
		(Index:=16#6072,	SubIndex:=0,		ValueType:=TYPE_UINT,		Access:=ACCESS_RW,	Eeprom:=EEPROM_NO,	AmpType:=BOTH_ROT_LIN,	WhenEnabled:=ENABLED_IMMEDIATELY),
		(Index:=16#6074,	SubIndex:=0,		ValueType:=TYPE_INT,		Access:=ACCESS_RO,		Eeprom:=EEPROM_NO,	AmpType:=BOTH_ROT_LIN,	WhenEnabled:=ENABLED_IMMEDIATELY),
		(Index:=16#6076,	SubIndex:=0,		ValueType:=TYPE_UDINT,		Access:=ACCESS_RO,		Eeprom:=EEPROM_NO,	AmpType:=BOTH_ROT_LIN,	WhenEnabled:=ENABLED_IMMEDIATELY),
		(Index:=16#6077,	SubIndex:=0,		ValueType:=TYPE_INT,		Access:=ACCESS_RO,		Eeprom:=EEPROM_NO,	AmpType:=BOTH_ROT_LIN,	WhenEnabled:=ENABLED_IMMEDIATELY),
		(Index:=16#607A,	SubIndex:=0,		ValueType:=TYPE_DINT,		Access:=ACCESS_RW,	Eeprom:=EEPROM_NO,	AmpType:=BOTH_ROT_LIN,	WhenEnabled:=ENABLED_IMMEDIATELY),
		(Index:=16#607C,	SubIndex:=0,		ValueType:=TYPE_DINT,		Access:=ACCESS_RW,	Eeprom:=EEPROM_YES,	AmpType:=BOTH_ROT_LIN,	WhenEnabled:=ENABLED_IMMEDIATELY),
(*330*)	(Index:=16#607D,	SubIndex:=0,		ValueType:=TYPE_USINT,		Access:=ACCESS_RO,		Eeprom:=EEPROM_NO,	AmpType:=BOTH_ROT_LIN,	WhenEnabled:=ENABLED_IMMEDIATELY),
		(Index:=16#607D,	SubIndex:=1,		ValueType:=TYPE_DINT,		Access:=ACCESS_RW,	Eeprom:=EEPROM_YES,	AmpType:=BOTH_ROT_LIN,	WhenEnabled:=ENABLED_IMMEDIATELY),
		(Index:=16#607D,	SubIndex:=2,		ValueType:=TYPE_DINT,		Access:=ACCESS_RW,	Eeprom:=EEPROM_YES,	AmpType:=BOTH_ROT_LIN,	WhenEnabled:=ENABLED_IMMEDIATELY),
		(Index:=16#607F,	SubIndex:=0,		ValueType:=TYPE_UDINT,		Access:=ACCESS_RW,	Eeprom:=EEPROM_YES,	AmpType:=BOTH_ROT_LIN,	WhenEnabled:=ENABLED_IMMEDIATELY),
		(Index:=16#6081,	SubIndex:=0,		ValueType:=TYPE_UDINT,		Access:=ACCESS_RW,	Eeprom:=EEPROM_YES,	AmpType:=BOTH_ROT_LIN,	WhenEnabled:=ENABLED_IMMEDIATELY),
		(Index:=16#6083,	SubIndex:=0,		ValueType:=TYPE_UDINT,		Access:=ACCESS_RW,	Eeprom:=EEPROM_YES,	AmpType:=BOTH_ROT_LIN,	WhenEnabled:=ENABLED_IMMEDIATELY),
		(Index:=16#6084,	SubIndex:=0,		ValueType:=TYPE_UDINT,		Access:=ACCESS_RW,	Eeprom:=EEPROM_YES,	AmpType:=BOTH_ROT_LIN,	WhenEnabled:=ENABLED_IMMEDIATELY),
		(Index:=16#6085,	SubIndex:=0,		ValueType:=TYPE_UDINT,		Access:=ACCESS_RW,	Eeprom:=EEPROM_YES,	AmpType:=BOTH_ROT_LIN,	WhenEnabled:=ENABLED_IMMEDIATELY),
		(Index:=16#6087,	SubIndex:=0,		ValueType:=TYPE_UDINT,		Access:=ACCESS_RW,	Eeprom:=EEPROM_YES,	AmpType:=BOTH_ROT_LIN,	WhenEnabled:=ENABLED_IMMEDIATELY),
		(Index:=16#6098,	SubIndex:=0,		ValueType:=TYPE_SINT,		Access:=ACCESS_RW,	Eeprom:=EEPROM_NO,	AmpType:=BOTH_ROT_LIN,	WhenEnabled:=ENABLED_IMMEDIATELY),
(*340*)	(Index:=16#6099,	SubIndex:=0,		ValueType:=TYPE_USINT,		Access:=ACCESS_RO,		Eeprom:=EEPROM_NO,	AmpType:=BOTH_ROT_LIN,	WhenEnabled:=ENABLED_IMMEDIATELY),
		(Index:=16#6099,	SubIndex:=1,		ValueType:=TYPE_UDINT,		Access:=ACCESS_RW,	Eeprom:=EEPROM_YES,	AmpType:=BOTH_ROT_LIN,	WhenEnabled:=ENABLED_IMMEDIATELY),
		(Index:=16#6099,	SubIndex:=2,		ValueType:=TYPE_UDINT,		Access:=ACCESS_RW,	Eeprom:=EEPROM_YES,	AmpType:=BOTH_ROT_LIN,	WhenEnabled:=ENABLED_IMMEDIATELY),
		(Index:=16#609A,	SubIndex:=0,		ValueType:=TYPE_UDINT,		Access:=ACCESS_RW,	Eeprom:=EEPROM_YES,	AmpType:=BOTH_ROT_LIN,	WhenEnabled:=ENABLED_IMMEDIATELY),
		(Index:=16#60B1,	SubIndex:=0,		ValueType:=TYPE_DINT,		Access:=ACCESS_RW,	Eeprom:=EEPROM_NO,	AmpType:=BOTH_ROT_LIN,	WhenEnabled:=ENABLED_IMMEDIATELY),
		(Index:=16#60B2,	SubIndex:=0,		ValueType:=TYPE_INT,		Access:=ACCESS_RW,	Eeprom:=EEPROM_NO,	AmpType:=BOTH_ROT_LIN,	WhenEnabled:=ENABLED_IMMEDIATELY),
		(Index:=16#60B8,	SubIndex:=0,		ValueType:=TYPE_UINT,		Access:=ACCESS_RW,	Eeprom:=EEPROM_NO,	AmpType:=BOTH_ROT_LIN,	WhenEnabled:=ENABLED_IMMEDIATELY),
		(Index:=16#60B9,	SubIndex:=0,		ValueType:=TYPE_UINT,		Access:=ACCESS_RO,		Eeprom:=EEPROM_NO,	AmpType:=BOTH_ROT_LIN,	WhenEnabled:=ENABLED_IMMEDIATELY),
		(Index:=16#60BA,	SubIndex:=0,		ValueType:=TYPE_DINT,		Access:=ACCESS_RO,		Eeprom:=EEPROM_NO,	AmpType:=BOTH_ROT_LIN,	WhenEnabled:=ENABLED_IMMEDIATELY),
		(Index:=16#60BC,	SubIndex:=0,		ValueType:=TYPE_DINT,		Access:=ACCESS_RO,		Eeprom:=EEPROM_NO,	AmpType:=BOTH_ROT_LIN,	WhenEnabled:=ENABLED_IMMEDIATELY),
(*350*)	(Index:=16#60C1,	SubIndex:=0,		ValueType:=TYPE_USINT,		Access:=ACCESS_RO,		Eeprom:=EEPROM_NO,	AmpType:=BOTH_ROT_LIN,	WhenEnabled:=ENABLED_IMMEDIATELY),
		(Index:=16#60C1,	SubIndex:=1,		ValueType:=TYPE_DINT,		Access:=ACCESS_RW,	Eeprom:=EEPROM_NO,	AmpType:=BOTH_ROT_LIN,	WhenEnabled:=ENABLED_IMMEDIATELY),
		(Index:=16#60C2,	SubIndex:=0,		ValueType:=TYPE_USINT,		Access:=ACCESS_RO,		Eeprom:=EEPROM_NO,	AmpType:=BOTH_ROT_LIN,	WhenEnabled:=ENABLED_IMMEDIATELY),
		(Index:=16#60C2,	SubIndex:=1,		ValueType:=TYPE_USINT,		Access:=ACCESS_RW,	Eeprom:=EEPROM_NO,	AmpType:=BOTH_ROT_LIN,	WhenEnabled:=ENABLED_IMMEDIATELY,		SpecialParameter:=CHANGE_ECAT_DISABLED),
		(Index:=16#60C2,	SubIndex:=2,		ValueType:=TYPE_SINT,		Access:=ACCESS_RW,	Eeprom:=EEPROM_NO,	AmpType:=BOTH_ROT_LIN,	WhenEnabled:=ENABLED_IMMEDIATELY,		SpecialParameter:=CHANGE_ECAT_DISABLED),
		(Index:=16#60E0,	SubIndex:=0,		ValueType:=TYPE_UINT,		Access:=ACCESS_RW,	Eeprom:=EEPROM_YES,	AmpType:=BOTH_ROT_LIN,	WhenEnabled:=ENABLED_IMMEDIATELY),
		(Index:=16#60E1,	SubIndex:=0,		ValueType:=TYPE_UINT,		Access:=ACCESS_RW,	Eeprom:=EEPROM_YES,	AmpType:=BOTH_ROT_LIN,	WhenEnabled:=ENABLED_IMMEDIATELY),
		(Index:=16#60F4,	SubIndex:=0,		ValueType:=TYPE_DINT,		Access:=ACCESS_RO,		Eeprom:=EEPROM_NO,	AmpType:=BOTH_ROT_LIN,	WhenEnabled:=ENABLED_IMMEDIATELY),
		(Index:=16#60FC,	SubIndex:=0,		ValueType:=TYPE_DINT,		Access:=ACCESS_RO,		Eeprom:=EEPROM_NO,	AmpType:=BOTH_ROT_LIN,	WhenEnabled:=ENABLED_IMMEDIATELY),
		(Index:=16#60FD,	SubIndex:=0,		ValueType:=TYPE_UDINT,		Access:=ACCESS_RO,		Eeprom:=EEPROM_NO,	AmpType:=BOTH_ROT_LIN,	WhenEnabled:=ENABLED_IMMEDIATELY),
(*360*)	(Index:=16#60FE,	SubIndex:=0,		ValueType:=TYPE_USINT,		Access:=ACCESS_RO,		Eeprom:=EEPROM_NO,	AmpType:=BOTH_ROT_LIN,	WhenEnabled:=ENABLED_IMMEDIATELY),
		(Index:=16#60FE,	SubIndex:=1,		ValueType:=TYPE_UDINT,		Access:=ACCESS_RW,	Eeprom:=EEPROM_NO,	AmpType:=BOTH_ROT_LIN,	WhenEnabled:=ENABLED_IMMEDIATELY),
		(Index:=16#60FE,	SubIndex:=2,		ValueType:=TYPE_UDINT,		Access:=ACCESS_RW,	Eeprom:=EEPROM_YES,	AmpType:=BOTH_ROT_LIN,	WhenEnabled:=ENABLED_IMMEDIATELY),
		(Index:=16#60FF,	SubIndex:=0,		ValueType:=TYPE_DINT,		Access:=ACCESS_RW,	Eeprom:=EEPROM_NO,	AmpType:=BOTH_ROT_LIN,	WhenEnabled:=ENABLED_IMMEDIATELY),
(*364*)	(Index:=16#6502,	SubIndex:=0,		ValueType:=TYPE_UDINT,		Access:=ACCESS_RO,		Eeprom:=EEPROM_NO,	AmpType:=BOTH_ROT_LIN,	WhenEnabled:=ENABLED_IMMEDIATELY)]
;
(*Internal variables*)
	State			:	UINT	:= 	0;
	Row				:	UINT	:= 	1;
	AmpType		:	UINT	;
	AmpVersion		:	UINT	;
	MaxRows		: 	UINT	:=	364;			(*If this is changed, also need to change array size*)
	(*FW 2 has 1 additional prm, but the prm is mirrored with an existing one, so no need to implement or change max rows *)
	FbVersion		:	UDINT	:=	Y_FB_VER_2_0;	(*Increase this with each revision of the function block*) (*Vers Up*)
	VendorID		: 	UDINT	;
	ProductCode		: 	UDINT	;
	RevisionNumber	: 	UDINT	;
	ProductName		:	STRING	;
	bNotExecute		:	BOOL	;

(*Internal Function Blocks*)
	fbRisingEdge			: 	R_TRIG	;
	fbFallingEdge		: 	F_TRIG	;

	fbFileBuffer 			:	FB_FileRingBuffer := (cbBuffer:=80000);	(*cbBuffer := 16#80000000, 2GB*)

	fbSdoReadExUint		: 	FB_EcCoESdoReadEx := (bCompleteAccess := FALSE);
	fbSdoReadExUdint	: 	FB_EcCoESdoReadEx := (bCompleteAccess := FALSE);
	fbSdoReadExUsint	: 	FB_EcCoESdoReadEx := (bCompleteAccess := FALSE);
	fbSdoReadExSint		: 	FB_EcCoESdoReadEx := (bCompleteAccess := FALSE);
	fbSdoReadExInt		: 	FB_EcCoESdoReadEx := (bCompleteAccess := FALSE);
	fbSdoReadExDint		: 	FB_EcCoESdoReadEx := (bCompleteAccess := FALSE);
	fbSdoReadExString	: 	FB_EcCoESdoReadEx := (bCompleteAccess := FALSE);

	fbLocalSystemTime	: 	FB_LocalSystemTime;

	systemTime			:	TIMESTRUCT	;
	bValidSystemTime	:	BOOL			;
	bEnableSystemTime	:	BOOL			;

	nErrorIDRead			:	UDINT			;
	sFileString			:	T_MaxString		;
	sNetIdRead			:	T_AmsNetId		;
	nSlaveAddrRead		:	UINT			;
	sFileRead			:	T_MaxString		;
	bBypassCheckRead	:	BOOL			;

END_VAR

fbFallingEdge	(CLK:= bExecute);
IF fbFallingEdge.Q THEN
	bNotExecute	:=	TRUE;
END_IF;

(* Done is TRUE for one cycle when falling edge of Execute has occured *)
IF bDone AND bNotExecute THEN
	bDone		:=	FALSE;
END_IF;

IF bError AND bNotExecute THEN
	bError				:=	FALSE;
	nErrorId				:=	0;
	nErrorIDRead			:=	0;
END_IF;

CASE State OF
0:
fbRisingEdge		(CLK:= bExecute);
IF fbRisingEdge.Q THEN
	bDone				:=	FALSE;
	bBusy				:=	TRUE;
	bError				:=	FALSE;
	nErrorId				:=	0;
	nErrorIDRead			:=	0;
	sErrorString			:=	'';
	sFileString			:=	sFileAuto;
	bNotExecute			:=	FALSE;
	sNetIdRead			:=	sNetId;
	nSlaveAddrRead		:=	nSlaveAddr;
	sFileRead			:=	sFile;
	bBypassCheckRead	:=	bBypassCheck;
	State				:=	1;
	Row					:=	1;
END_IF

1:
fbSdoReadExUdint(
	sNetId		:=	sNetIdRead,
	nSlaveAddr	:=	nSlaveAddrRead,
	nIndex		:=	16#1018,
	nSubIndex	:=	1,				(*Vendor ID*)
	pDstBuf		:=	ADR(VendorID),
	cbBufLen	:=	SIZEOF(VendorID),
	bExecute	:=	FALSE	);
fbLocalSystemTime(					(*Used for file name*)
	bEnable		:=	FALSE,
	bValid=>bValidSystemTime);
State:=2;

2:
fbSdoReadExUdint(bExecute:= TRUE);
State:=3;

3: (*SDO read, Read ID*)
fbSdoReadExUdint();
IF NOT fbSdoReadExUdint.bBusy THEN
	IF NOT fbSdoReadExUdint.bError THEN
		fbSdoReadExUdint(bExecute:= FALSE);
		State:=4;
		IF NOT (VendorID=VENDOR_YASKAWA) THEN 			(*Vendor ID = Yaskawa*)
			sErrorString:=CONCAT(CONCAT(
				'Product not compatible.  This FB is only for Vendor ID 0x00000539 (Yaskawa).  Vendor ID read as ',
				UDINT_TO_STRING(VendorID)),
				'.  ErrorID from FB, not from ADS.'
			);
			nErrorIDRead:=4100;
			State:=99;
		END_IF
	ELSE
		sErrorString:=CONCAT(CONCAT(
			'Error reading Product Code, Object: ',
			WORD_TO_STRING(fbSdoReadExUdint.nIndex)),
			'.  Error occurred using Function Block FB_EcCoESdoReadEx for UDINT.  ErrorID is from FB_EcCoESdoReadEx.'
		);
		nErrorIDRead:=fbSdoReadExUdint.nErrId;
		State:=99;
	END_IF
END_IF

4:
fbSdoReadExUdint(
	nSubIndex	:=	2,				(*Product Code*)
	pDstBuf		:=	ADR(ProductCode),
	cbBufLen	:=	SIZEOF(ProductCode),
	bExecute	:=	TRUE);
State:=5;

5: (*SDO read, Read ID*)
fbSdoReadExUdint();
IF NOT fbSdoReadExUdint.bBusy THEN
	IF NOT fbSdoReadExUdint.bError THEN
		fbSdoReadExUdint(bExecute:= FALSE);
		State:=6;
		IF ProductCode=PRODUCT_ROTARY THEN 			(*Rotary Motor Detected*)
			AmpType		:= ROTARY;
		ELSE IF ProductCode=PRODUCT_LINEAR THEN 	(*Linear Motor Detected*)
			AmpType		:= LINEAR;
		ELSE 									 (*neither Linear nor Rotary Motor Detected*)
			sErrorString:=CONCAT(CONCAT(
				'Product not compatible.  This FB is only for Product codes 0x02200001 (Sigma-5 Rotary) and 0x02200002 (Sigma-5 Linear).  If using Sigma-5 CoE Drive, get latest FB from Yaskawa.com.  Product code read as ',
				UDINT_TO_STRING(ProductCode)),
				'.  ErrorID from FB, not from ADS.'
			);
			nErrorIDRead:=4101;
			State:=99;
		END_IF
		END_IF
	ELSE
		sErrorString:=CONCAT(CONCAT(
			'Error reading Product Code, Object: ',
			WORD_TO_STRING(fbSdoReadExUdint.nIndex)),
			'.  Error occurred using Function Block FB_EcCoESdoReadEx for UDINT.  ErrorID is from FB_EcCoESdoReadEx.'
		);
		nErrorIDRead:=fbSdoReadExUdint.nErrId;
		State:=99;
	END_IF
END_IF

6:
fbSdoReadExUdint(
	nSubIndex	:=	3,				(*Revision Number*)
	pDstBuf		:=	ADR(RevisionNumber),
	cbBufLen	:=	SIZEOF(RevisionNumber),
	bExecute	:=	TRUE);
State:=7;

7:
fbSdoReadExUdint();
IF NOT fbSdoReadExUdint.bBusy THEN
	IF NOT fbSdoReadExUdint.bError THEN
		fbSdoReadExUdint(bExecute:= FALSE);
		State:=8;
		IF RevisionNumber=REVISION_1 THEN 			(*Version 1.0*) (*IF statement to allow future version implementations*)
			AmpVersion		:= VERS_1_0;
		ELSE IF RevisionNumber=REVISION_2 THEN		(*Vers Up*)
			AmpVersion		:= VERS_2_0;				(*Vers Up*)
		ELSE 									 (*neither Linear nor Rotary Motor Detected*)
			IF NOT bBypassCheckRead THEN
				sErrorString:=CONCAT(CONCAT(
(*Vers Up*)			'Product not compatible.  This FB is only for Revision Number 0x00010000 (Vers.1.0) or 0x00020000 (Vers.2.0).  If using Sigma-5 CoE Drive, get latest FB from Yaskawa.com.  Revision Number read as ',
					UDINT_TO_STRING(RevisionNumber)),
					'.  ErrorID from FB, not from ADS.'
				);
				nErrorIDRead:=4102;
				State:=99;
			END_IF
		END_IF
		END_IF			(*Vers Up*)
	ELSE
		sErrorString:=CONCAT(CONCAT(
			'Error reading Product Code, Object: ',
			WORD_TO_STRING(fbSdoReadExUdint.nIndex)),
			'.  Error occurred using Function Block FB_EcCoESdoReadEx for UDINT.  ErrorID is from FB_EcCoESdoReadEx.'
		);
		nErrorIDRead:=fbSdoReadExUdint.nErrId;
		State:=99;
	END_IF
END_IF

8:
fbSdoReadExSint(
	sNetId		:= sNetIdRead,
	nSlaveAddr	:= nSlaveAddrRead,
	bExecute	:= FALSE	);
fbSdoReadExInt(
	sNetId		:= sNetIdRead,
	nSlaveAddr	:= nSlaveAddrRead,
	bExecute	:= FALSE	);
fbSdoReadExDint(
	sNetId		:= sNetIdRead,
	nSlaveAddr	:= nSlaveAddrRead,
	bExecute	:= FALSE	);
fbSdoReadExUsint(
	sNetId		:= sNetIdRead,
	nSlaveAddr	:= nSlaveAddrRead,
	bExecute	:= FALSE	);
fbSdoReadExUint(
	sNetId		:= sNetIdRead,
	nSlaveAddr	:= nSlaveAddrRead,
	bExecute	:= FALSE	);
fbSdoReadExUdint(); (*already false and initialized from above*)
fbSdoReadExString(
	sNetId		:= sNetIdRead,
	nSlaveAddr	:= nSlaveAddrRead,
	bExecute	:= FALSE	);
State:=10;

10:
IF NOT (Row=MaxRows+1) THEN
	IF AllSigmaObjects[Row].AmpType=BOTH_ROT_LIN OR AllSigmaObjects[Row].AmpType=AmpType THEN (*If parameter set is for either rotary/linear, or parameter set is for just rotary or just linear*)
		CASE AllSigmaObjects[Row].ValueType OF
		TYPE_SINT:
			fbSdoReadExSint(
				nIndex		:= AllSigmaObjects[Row].Index,
				nSubIndex	:= AllSigmaObjects[Row].SubIndex,
				pDstBuf		:= ADR(AllSigmaObjects[Row].ValueSint),
				cbBufLen	:= SIZEOF(AllSigmaObjects[Row].ValueSint),
				bExecute	:= TRUE );
			State:=20;
		TYPE_INT:
			fbSdoReadExInt(
				nIndex		:= AllSigmaObjects[Row].Index,
				nSubIndex	:= AllSigmaObjects[Row].SubIndex,
				pDstBuf		:= ADR(AllSigmaObjects[Row].ValueInt),
				cbBufLen	:= SIZEOF(AllSigmaObjects[Row].ValueInt),
				bExecute	:= TRUE );
			State:=30;
		TYPE_DINT:
			fbSdoReadExDint(
				nIndex		:= AllSigmaObjects[Row].Index,
				nSubIndex	:= AllSigmaObjects[Row].SubIndex,
				pDstBuf		:= ADR(AllSigmaObjects[Row].ValueDint),
				cbBufLen	:= SIZEOF(AllSigmaObjects[Row].ValueDint),
				bExecute	:= TRUE );
			State:=40;
		TYPE_USINT:
			fbSdoReadExUsint(
				nIndex		:= AllSigmaObjects[Row].Index,
				nSubIndex	:= AllSigmaObjects[Row].SubIndex,
				pDstBuf		:= ADR(AllSigmaObjects[Row].ValueUsint),
				cbBufLen	:= SIZEOF(AllSigmaObjects[Row].ValueUsint),
				bExecute	:= TRUE );
			State:=50;
		TYPE_UINT:
			fbSdoReadExUint(
				nIndex		:= AllSigmaObjects[Row].Index,
				nSubIndex	:= AllSigmaObjects[Row].SubIndex,
				pDstBuf		:= ADR(AllSigmaObjects[Row].ValueUint),
				cbBufLen	:= SIZEOF(AllSigmaObjects[Row].ValueUint),
				bExecute	:= TRUE );
			State:=60;
		TYPE_UDINT:
			fbSdoReadExUdint(
				nIndex		:= AllSigmaObjects[Row].Index,
				nSubIndex	:= AllSigmaObjects[Row].SubIndex,
				pDstBuf		:= ADR(AllSigmaObjects[Row].ValueUdint),
				cbBufLen	:= SIZEOF(AllSigmaObjects[Row].ValueUdint),
				bExecute	:= TRUE );
			State:=70;
		TYPE_STRING:
			fbSdoReadExString(
				nIndex		:= AllSigmaObjects[Row].Index,
				nSubIndex	:= AllSigmaObjects[Row].SubIndex,
				pDstBuf		:= ADR(AllSigmaObjects[Row].ValueString),
				cbBufLen	:= SIZEOF(AllSigmaObjects[Row].ValueString),
				bExecute	:= TRUE );
			State:=80;

		ELSE
			sErrorString:=CONCAT(CONCAT(
				'Error reading Object Data Type or Data Type not supported.  Enumerated value read as: ',
				USINT_TO_STRING(AllSigmaObjects[Row].ValueType)),
				'.'
			);
			nErrorIDRead:=4103;
			State:=99;
		END_CASE

	ELSE
		Row:=Row+1;
	END_IF
ELSE
	State:=100;
	IF bBypassAutoFile THEN
		State:=110;
	END_IF
END_IF

20: (*Read SINT*)
fbSdoReadExSint();
IF NOT fbSdoReadExSint.bBusy THEN
	IF NOT fbSdoReadExSint.bError THEN
		Row:=Row+1;
		fbSdoReadExSint(bExecute:= FALSE);
		State:=10;
	ELSE
		sErrorString:=CONCAT(CONCAT(
			'Error reading CoE Object ',
			WORD_TO_STRING(AllSigmaObjects[Row].Index)),
			'.  Error occurred using Function Block FB_EcCoESdoReadEx for SINT.  ErrorID is from FB_EcCoESdoReadEx.'
		);
		nErrorIDRead:=fbSdoReadExSint.nErrId;
		State:=99;
	END_IF
END_IF

30: (*Read INT*)
fbSdoReadExInt();
IF NOT fbSdoReadExInt.bBusy THEN
	IF NOT fbSdoReadExInt.bError THEN
		Row:=Row+1;
		fbSdoReadExInt(bExecute:= FALSE);
		State:=10;
	ELSE
		sErrorString:=CONCAT(CONCAT(
			'Error reading CoE Object ',
			WORD_TO_STRING(AllSigmaObjects[Row].Index)),
			'.  Error occurred using Function Block FB_EcCoESdoReadEx for INT.  ErrorID is from FB_EcCoESdoReadEx.'
		);
		nErrorIDRead:=fbSdoReadExInt.nErrId;
		State:=99;
	END_IF
END_IF

40: (*Read DINT*)
fbSdoReadExDint();
IF NOT fbSdoReadExDint.bBusy THEN
	IF NOT fbSdoReadExDint.bError THEN
		Row:=Row+1;
		fbSdoReadExDint(bExecute:= FALSE);
		State:=10;
	ELSE
		sErrorString:=CONCAT(CONCAT(
			'Error reading CoE Object ',
			WORD_TO_STRING(AllSigmaObjects[Row].Index)),
			'.  Error occurred using Function Block FB_EcCoESdoReadEx for DINT.  ErrorID is from FB_EcCoESdoReadEx.'
		);
		nErrorIDRead:=fbSdoReadExDint.nErrId;
		State:=99;
	END_IF
END_IF

50: (*Read USINT*)
fbSdoReadExUsint();
IF NOT fbSdoReadExUsint.bBusy THEN
	IF NOT fbSdoReadExUsint.bError THEN
		Row:=Row+1;
		fbSdoReadExUsint(bExecute:= FALSE);
		State:=10;
	ELSE
		sErrorString:=CONCAT(CONCAT(
			'Error reading CoE Object ',
			WORD_TO_STRING(AllSigmaObjects[Row].Index)),
			'.  Error occurred using Function Block FB_EcCoESdoReadEx for USINT.  ErrorID is from FB_EcCoESdoReadEx.'
		);
		nErrorIDRead:=fbSdoReadExUsint.nErrId;
		State:=99;
	END_IF
END_IF

60: (*Read UINT*)
fbSdoReadExUint();
IF NOT fbSdoReadExUint.bBusy THEN
	IF NOT fbSdoReadExUint.bError THEN
		Row:=Row+1;
		fbSdoReadExUint(bExecute:= FALSE);
		State:=10;
	ELSE
		sErrorString:=CONCAT(CONCAT(
			'Error reading CoE Object ',
			WORD_TO_STRING(AllSigmaObjects[Row].Index)),
			'.  Error occurred using Function Block FB_EcCoESdoReadEx for UINT.  ErrorID is from FB_EcCoESdoReadEx.'
		);
		nErrorIDRead:=fbSdoReadExUint.nErrId;
		State:=99;
	END_IF
END_IF

70: (*Read UDINT*)
fbSdoReadExUdint();
IF NOT fbSdoReadExUdint.bBusy THEN
	IF NOT fbSdoReadExUdint.bError THEN
		Row:=Row+1;
		fbSdoReadExUdint(bExecute:= FALSE);
		State:=10;
	ELSE
		sErrorString:=CONCAT(CONCAT(
			'Error reading CoE Object ',
			WORD_TO_STRING(AllSigmaObjects[Row].Index)),
			'.  Error occurred using Function Block FB_EcCoESdoReadEx for UDINT.  ErrorID is from FB_EcCoESdoReadEx.'
		);
		nErrorIDRead:=fbSdoReadExUdint.nErrId;
		State:=99;
	END_IF
END_IF

80: (*Read STRING*)
fbSdoReadExString();
IF NOT fbSdoReadExString.bBusy THEN
	IF NOT fbSdoReadExString.bError THEN
		Row:=Row+1;
		fbSdoReadExString(bExecute:= FALSE);
		State:=10;
	ELSE
		sErrorString:=CONCAT(CONCAT(
			'Error reading CoE Object ',
			WORD_TO_STRING(AllSigmaObjects[Row].Index)),
			'.  Error occurred using Function Block FB_EcCoESdoReadEx for STRING.  ErrorID is from FB_EcCoESdoReadEx.'
		);
		nErrorIDRead:=fbSdoReadExString.nErrId;
		State:=99;
	END_IF
END_IF

100:
fbLocalSystemTime(
	bEnable:= TRUE,
	bValid=>bValidSystemTime,
	systemTime=> systemTime);

fbFileBuffer(nID		:=	FbVersion);
IF NOT fbFileBuffer.bBusy AND bValidSystemTime THEN (*just in case file buffer is busy from a previous call*)
		sFileString:=CONCAT(sFileAuto,AllSigmaObjects[3].ValueString); (*Row 3 is object 1008*)
	IF AmpType=ROTARY THEN
		sFileString:=CONCAT(sFileString,'_Rot');
	ELSE
		sFileString:=CONCAT(sFileString,'_Lin');
	END_IF
	IF AmpVersion= VERS_1_0 THEN
		sFileString:=CONCAT(sFileString,'Ver1.0');
	ELSE IF AmpVersion= VERS_2_0 THEN			(*Vers Up*)
		sFileString:=CONCAT(sFileString,'Ver2.0');		(*Vers Up*)
	END_IF										(*Vers Up*)
	END_IF
	sFileString:=CONCAT(CONCAT(sFileString,'_Addr'),UINT_TO_STRING(nSlaveAddrRead));

	sFileString:=
		CONCAT(
		CONCAT(
		CONCAT(
		CONCAT(
		CONCAT(
		CONCAT(
			sFileString,
			'_'),
			WORD_TO_STRING(systemTime.wMonth)),
			'-'),
			WORD_TO_STRING(systemTime.wDay)),
			'-'),
			WORD_TO_STRING(systemTime.wYear));

	sFileString:=CONCAT(sFileString,'_');

	sFileString:=
		CONCAT(
		CONCAT(
		CONCAT(
		CONCAT(
		CONCAT(
		CONCAT(
			sFileString,
			WORD_TO_STRING(systemTime.wHour)),
			'.'),
			WORD_TO_STRING(systemTime.wMinute)),
			'.'),
			WORD_TO_STRING(systemTime.wSecond)),
			'.dat');
	fbFileBuffer.A_Create();					(*Open File on next call of fbFileBuffer*)
	State:=101;
END_IF

101:
fbFileBuffer(sPathName:=sFileString);
IF NOT fbFileBuffer.bBusy THEN
	IF NOT fbFileBuffer.bError THEN
		fbFileBuffer.A_AddTail(
			pWriteBuff	:= ADR(AllSigmaObjects),
			cbWriteLen	:= SIZEOF(AllSigmaObjects));
		State:=102;
	ELSE
		sErrorString:=CONCAT(CONCAT(
			'Error creating first file (the backup): ',
			sFileString),
			'.  Error occurred using Function Call FB_FileRingBuffer.A_Create.  ErrorID is from FB_FileRingBuffer.'
		);
		nErrorIDRead:=fbFileBuffer.nErrID;
		State:=99;
	END_IF
END_IF

102:
fbFileBuffer();
IF NOT fbFileBuffer.bBusy THEN
	IF NOT fbFileBuffer.bError THEN
		fbFileBuffer.A_Close();
		State:=110;
	ELSE
		sErrorString:=CONCAT(CONCAT(
			'Error writing Sigma Objects to File: ',
			sFileString),
			'.  Error occurred using Function Call FB_FileRingBuffer.A_AddTail.  ErrorID is from FB_FileRingBuffer.'
		);
		nErrorIDRead:=fbFileBuffer.nErrID;
		State:=99;
	END_IF
END_IF

110:(*File closed, Make a copy*)
fbFileBuffer(nID		:=	FbVersion);
IF NOT fbFileBuffer.bBusy THEN
	IF NOT fbFileBuffer.bError THEN
		fbFileBuffer.A_Create();
		State:=111;
	ELSE
		sErrorString:=CONCAT(CONCAT(
			'Error closing backup file: ',
			sFileString),
			'.  Error occurred using Function Call FB_FileRingBuffer.A_Close.  ErrorID is from FB_FileRingBuffer.'
		);
		nErrorIDRead:=fbFileBuffer.nErrID;
		State:=99;
	END_IF
END_IF

111:
fbFileBuffer(sPathName:=sFileRead);
IF NOT fbFileBuffer.bBusy THEN
	IF NOT fbFileBuffer.bError THEN
		fbFileBuffer.A_AddTail(
			pWriteBuff	:= ADR(AllSigmaObjects),
			cbWriteLen	:= SIZEOF(AllSigmaObjects));
			State:=112;
	ELSE
		sErrorString:=CONCAT(CONCAT(
			'Error creating second file (last read): ',
			sFileRead),
			'.  Error occurred using Function Call FB_FileRingBuffer.A_Create.  ErrorID is from FB_FileRingBuffer.'
		);
		nErrorIDRead:=fbFileBuffer.nErrID;
		State:=99;
	END_IF
END_IF

112:
fbFileBuffer();
IF NOT fbFileBuffer.bBusy THEN
	IF NOT fbFileBuffer.bError THEN
		fbFileBuffer.A_Close();
		State:=113;
	ELSE
		sErrorString:=CONCAT(CONCAT(
			'Error writing STRING Objects to second file (last read): ',
			sFileRead),
			'.  Error occurred using Function Call FB_FileRingBuffer.A_AddTail.  ErrorID is from FB_FileRingBuffer.'
		);
		nErrorIDRead:=fbFileBuffer.nErrID;
		State:=99;
	END_IF
END_IF

113: (*File closed*)
fbFileBuffer();
IF NOT fbFileBuffer.bBusy THEN
	IF NOT fbFileBuffer.bError THEN
		bDone	:=	TRUE;
		bBusy	:=	FALSE;
		State:=0;
	ELSE
		sErrorString:=CONCAT(CONCAT(
			'Error closing backup file: ',
			sFileRead),
			'.  Error occurred using Function Call FB_FileRingBuffer.A_Close.  ErrorID is from FB_FileRingBuffer.'
		);
		nErrorIDRead:=fbFileBuffer.nErrID;
		State:=99;
	END_IF
END_IF

99: (*Error State*)
	bBusy	:=	FALSE;
	bError	:=	TRUE;
	nErrorID	:=	nErrorIDRead;
	State	:=	0;
ELSE
;
END_CASE

END_FUNCTION_BLOCK

// POUs/Y_WriteParameters
FUNCTION_BLOCK Y_WriteParameters
VAR_INPUT
	bExecute	:	BOOL		;
	sNetId		:	T_AmsNetId	;
	nSlaveAddr 	:	UINT		;
	sFile		:	T_MaxString	:=	'C:\YaskawaPrm.dat';
END_VAR
VAR_OUTPUT
	bDone		:	BOOL	;
	bBusy		:	BOOL	;
	bError		:	BOOL	;
	nErrorID		:	UDINT	;
END_VAR
VAR
	(*Extra Features Var In*)
	bBypassCheck	:	BOOL		;					(*Used to skip Version check, but not Vendor ID nor Product Code*)
	(*Extra Features Var Out*)
	sErrorString		:	T_MaxString	;

	State				:	UINT		:= 	0;
	Row					:	UINT		:=	1;
	AmpType			:	UINT		;
	AmpVersion			:	UINT		;
	MaxRows			: 	UINT		:=	364;				(*If this is changed, also need to change array size*)
	AllSigmaObjects 		: 	ARRAY			[1..364] OF ST_SigmaObject;
	FbVersion			:	UDINT		:=	Y_FB_VER_2_0;	(*Increase this with each revision of the function block*)	(*Vers Up*)
	VendorID			: 	UDINT		;
	ProductCode			: 	UDINT		;
	RevisionNumber		: 	UDINT		;
	StatusWord			: 	UINT		;
	StorePrmStatus		:	UDINT		;
	PrmCfgStatus			:	UDINT		;
	bNotExecute			:	BOOL		;
	nErrorIDRead			:	UDINT		;
	sFileString			:	T_MaxString	;
	sNetIdRead			:	T_AmsNetId	;
	nSlaveAddrRead		:	UINT		;
	sFileRead			:	T_MaxString	;
	bBypassCheckRead	:	BOOL		;

(*Internal Function Blocks*)
	fbFileBuffer 			:	FB_FileRingBuffer			:= (cbBuffer := 80000);	(*cbBuffer := 16#80000000, 2GB*)

	fbRisingEdge			: 	R_TRIG	;
	fbFallingEdge		: 	F_TRIG	;

